(* Schneider Machine Expert - Basic project Controller3(2shkaf), file version 2.4.0.0 *)
(* ProjectInformations: Name=New project *)

HARDWARE
  Cpu 0: TM221CE40T
  ModuleExtensionObject 0: TM3DI32K
  ModuleExtensionObject 1: TM3DI32K
  ModuleExtensionObject 2: TM3DI32K
  ModuleExtensionObject 3: TM3DI32K
  ModuleExtensionObject 4: TM3DI32K
  ModuleExtensionObject 5: TM3DQ32TK
  ModuleExtensionObject 6: TM3DQ32TK
  Cartridge1 0: TMC2SL1
  EthernetConfiguration: NetworkName=M221, IpAllocationMode=FixedAddress, IpAddress=192.168.1.202, SubnetMask=255.255.255.0
  EthernetConfiguration: NetworkName=M221, IpAllocationMode=FixedAddress, IpAddress=0.0.0.0, SubnetMask=0.0.0.0
  SerialLineConfiguration: Baud=Baud19200, Parity=ParityNone, DataBits=DataBits8, StopBits=StopBits1, PhysicalMedium=PhysicalMediumRs485, TransmissionMode=TransmissionModeModbusRtu, SlaveId=1, Addressing=MasterAddressing
  MastTask: UsePeriodScanMode=false, PeriodScan=100
  FastTask: Period=255
  CpuBehavior: StartingMode=StartAutoRunForced, AutoSaveRamOnEeprom=true, WatchdogPeriod=250

SYMBOLS  (address, symbol, comment, settings)
  %M0       SMS  "0_3"
  %TM0        [Preset=3, Base=OneSecond]
  %TM1        [Preset=3, Base=OneSecond]
  %TM2        [Preset=3, Base=OneSecond]
  %TM3        [Preset=3, Base=OneSecond]
  %TM4        [Preset=3, Base=OneSecond]
  %TM5        [Preset=3, Base=OneSecond]
  %TM6        [Preset=3, Base=OneSecond]
  %TM7        [Preset=3, Base=OneSecond]
  %TM8        [Preset=3, Base=OneSecond]
  %TM9        [Preset=3, Base=OneSecond]
  %TM10       [Preset=3, Base=OneSecond]
  %TM11       [Preset=3, Base=OneSecond]
  %TM12       [Preset=3, Base=OneSecond]
  %TM13       [Preset=3, Base=OneSecond]
  %TM14       [Preset=3, Base=OneSecond]
  %TM15       [Preset=3, Base=OneSecond]
  %TM16       [Preset=3, Base=OneSecond]
  %TM17       [Preset=3, Base=OneSecond]
  %TM18       [Preset=3, Base=OneSecond]
  %TM19       [Preset=3, Base=OneSecond]
  %TM20       [Preset=3, Base=OneSecond]
  %TM21       [Preset=3, Base=OneSecond]
  %TM22       [Preset=3, Base=OneSecond]
  %TM23       [Preset=3, Base=OneSecond]

POU Входы 2.0
  (* SectionNumber=1 *)

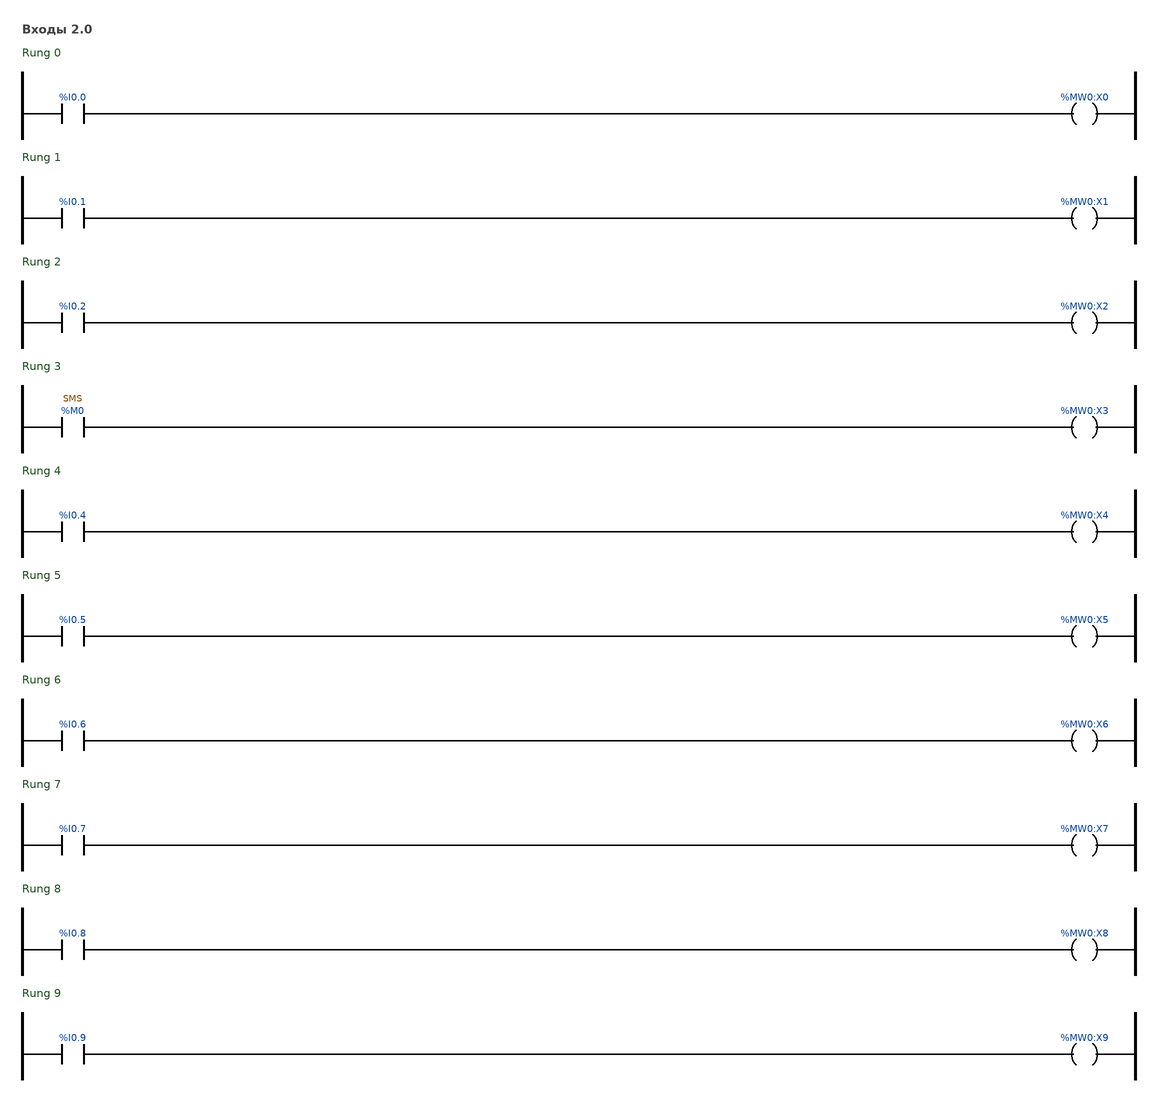

// Rung 0
  LD %I0.0
  ST %MW0:X0
  // as ST:
  //   %MW0:X0 := %I0.0;

// Rung 1
  LD %I0.1
  ST %MW0:X1
  // as ST:
  //   %MW0:X1 := %I0.1;

// Rung 2
  LD %I0.2
  ST %MW0:X2
  // as ST:
  //   %MW0:X2 := %I0.2;

// Rung 3
  LD %M0                  (* SMS *)
  ST %MW0:X3
  // as ST:
  //   %MW0:X3 := SMS;

// Rung 4
  LD %I0.4
  ST %MW0:X4
  // as ST:
  //   %MW0:X4 := %I0.4;

// Rung 5
  LD %I0.5
  ST %MW0:X5
  // as ST:
  //   %MW0:X5 := %I0.5;

// Rung 6
  LD %I0.6
  ST %MW0:X6
  // as ST:
  //   %MW0:X6 := %I0.6;

// Rung 7
  LD %I0.7
  ST %MW0:X7
  // as ST:
  //   %MW0:X7 := %I0.7;

// Rung 8
  LD %I0.8
  ST %MW0:X8
  // as ST:
  //   %MW0:X8 := %I0.8;

// Rung 9
  LD %I0.9
  ST %MW0:X9
  // as ST:
  //   %MW0:X9 := %I0.9;

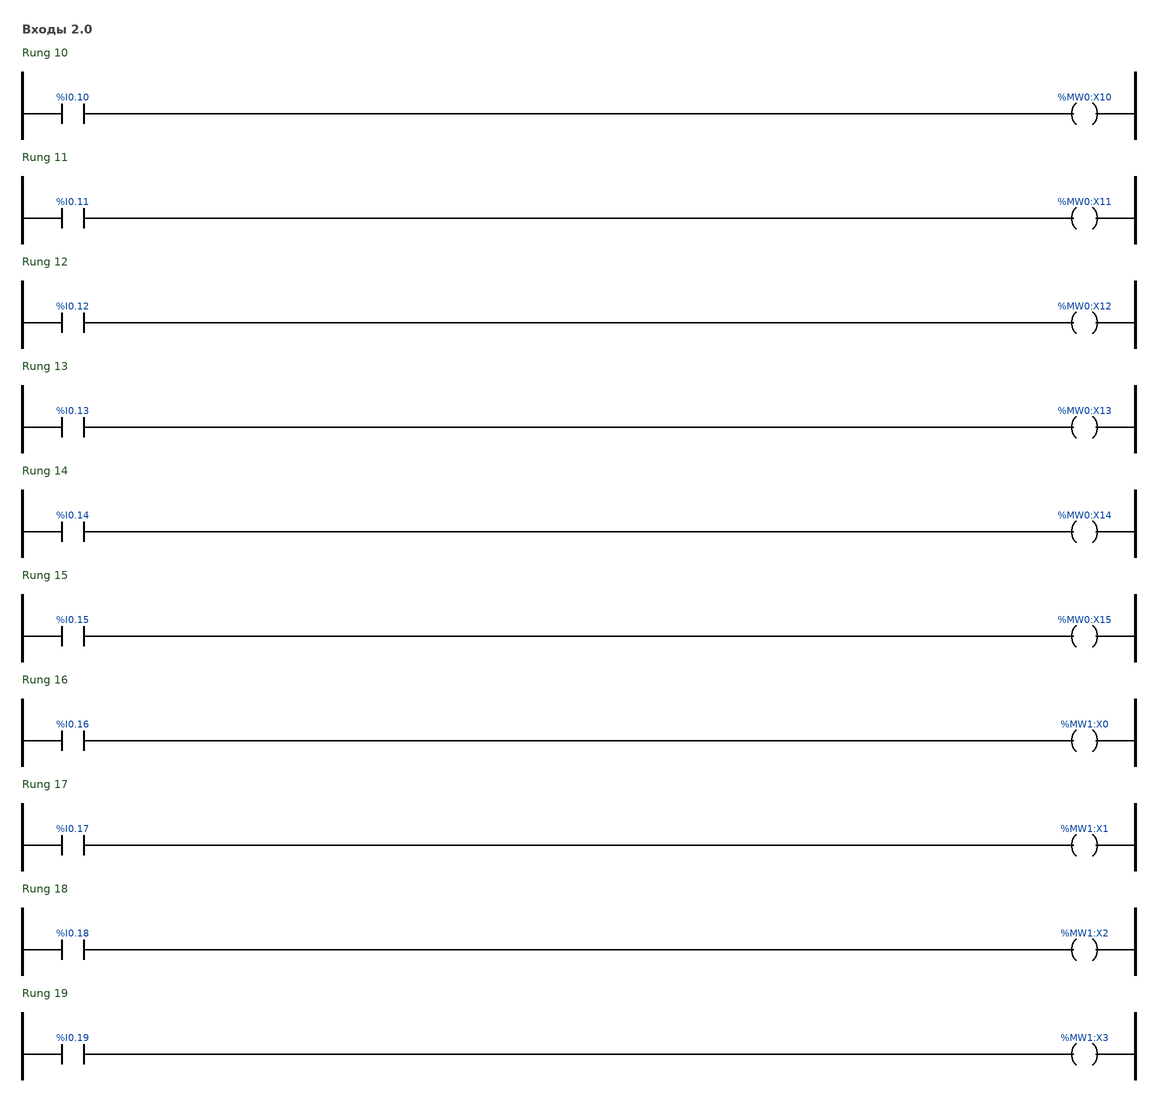

// Rung 10
  LD %I0.10
  ST %MW0:X10
  // as ST:
  //   %MW0:X10 := %I0.10;

// Rung 11
  LD %I0.11
  ST %MW0:X11
  // as ST:
  //   %MW0:X11 := %I0.11;

// Rung 12
  LD %I0.12
  ST %MW0:X12
  // as ST:
  //   %MW0:X12 := %I0.12;

// Rung 13
  LD %I0.13
  ST %MW0:X13
  // as ST:
  //   %MW0:X13 := %I0.13;

// Rung 14
  LD %I0.14
  ST %MW0:X14
  // as ST:
  //   %MW0:X14 := %I0.14;

// Rung 15
  LD %I0.15
  ST %MW0:X15
  // as ST:
  //   %MW0:X15 := %I0.15;

// Rung 16
  LD %I0.16
  ST %MW1:X0
  // as ST:
  //   %MW1:X0 := %I0.16;

// Rung 17
  LD %I0.17
  ST %MW1:X1
  // as ST:
  //   %MW1:X1 := %I0.17;

// Rung 18
  LD %I0.18
  ST %MW1:X2
  // as ST:
  //   %MW1:X2 := %I0.18;

// Rung 19
  LD %I0.19
  ST %MW1:X3
  // as ST:
  //   %MW1:X3 := %I0.19;

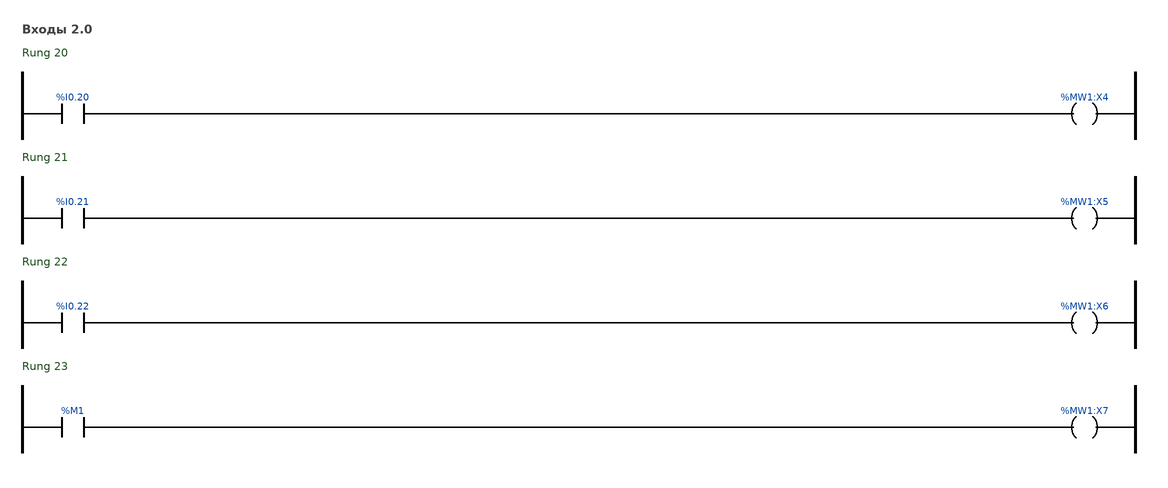

// Rung 20
  LD %I0.20
  ST %MW1:X4
  // as ST:
  //   %MW1:X4 := %I0.20;

// Rung 21
  LD %I0.21
  ST %MW1:X5
  // as ST:
  //   %MW1:X5 := %I0.21;

// Rung 22
  LD %I0.22
  ST %MW1:X6
  // as ST:
  //   %MW1:X6 := %I0.22;

// Rung 23
  LD %M1
  ST %MW1:X7
  // as ST:
  //   %MW1:X7 := %M1;

POU Входы 2.1
  (* SectionNumber=2 *)

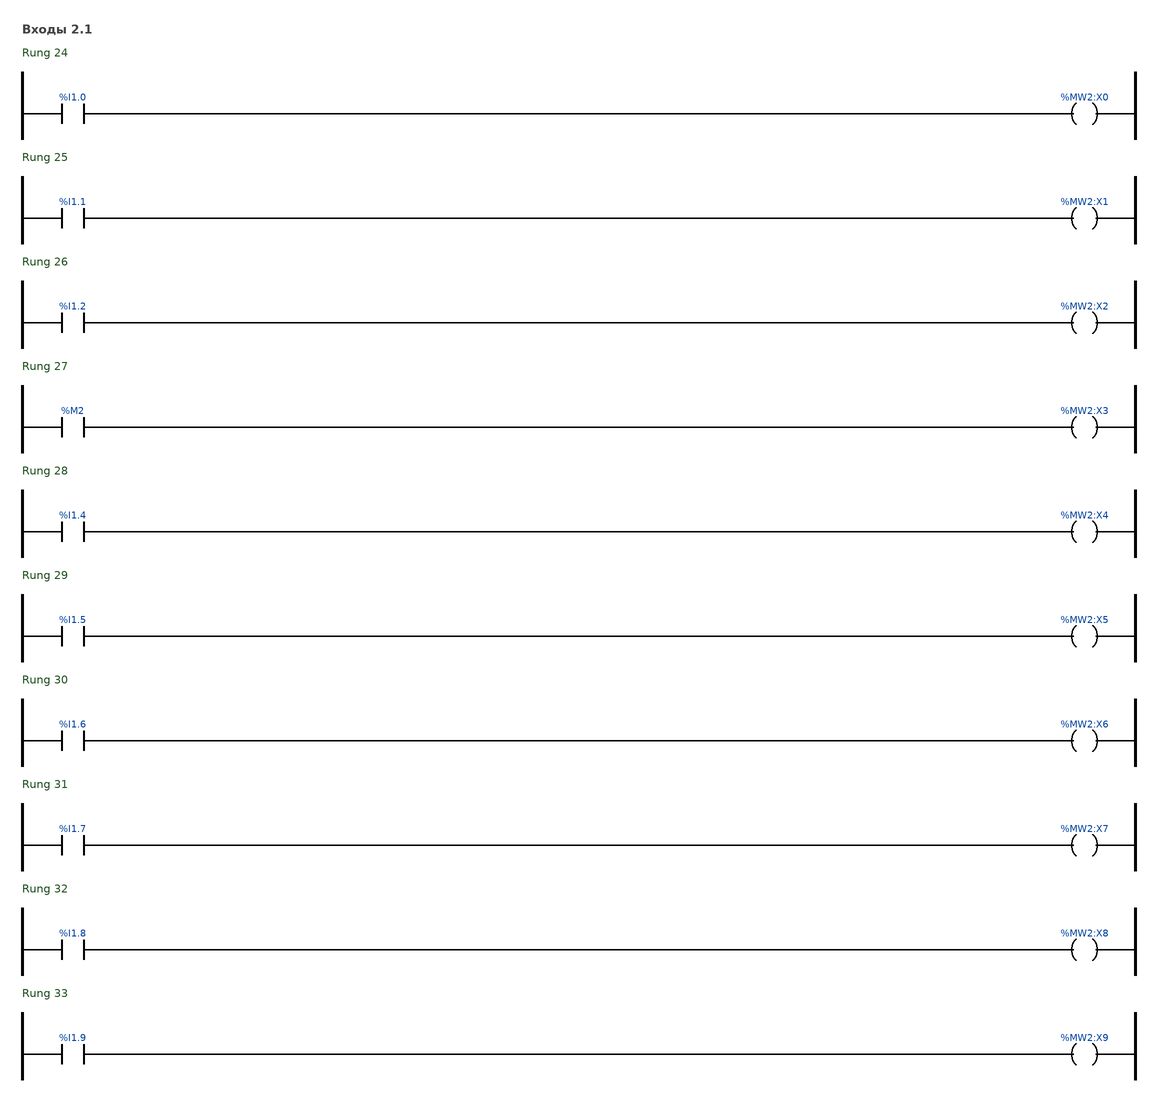

// Rung 24
  LD %I1.0
  ST %MW2:X0
  // as ST:
  //   %MW2:X0 := %I1.0;

// Rung 25
  LD %I1.1
  ST %MW2:X1
  // as ST:
  //   %MW2:X1 := %I1.1;

// Rung 26
  LD %I1.2
  ST %MW2:X2
  // as ST:
  //   %MW2:X2 := %I1.2;

// Rung 27
  LD %M2
  ST %MW2:X3
  // as ST:
  //   %MW2:X3 := %M2;

// Rung 28
  LD %I1.4
  ST %MW2:X4
  // as ST:
  //   %MW2:X4 := %I1.4;

// Rung 29
  LD %I1.5
  ST %MW2:X5
  // as ST:
  //   %MW2:X5 := %I1.5;

// Rung 30
  LD %I1.6
  ST %MW2:X6
  // as ST:
  //   %MW2:X6 := %I1.6;

// Rung 31
  LD %I1.7
  ST %MW2:X7
  // as ST:
  //   %MW2:X7 := %I1.7;

// Rung 32
  LD %I1.8
  ST %MW2:X8
  // as ST:
  //   %MW2:X8 := %I1.8;

// Rung 33
  LD %I1.9
  ST %MW2:X9
  // as ST:
  //   %MW2:X9 := %I1.9;

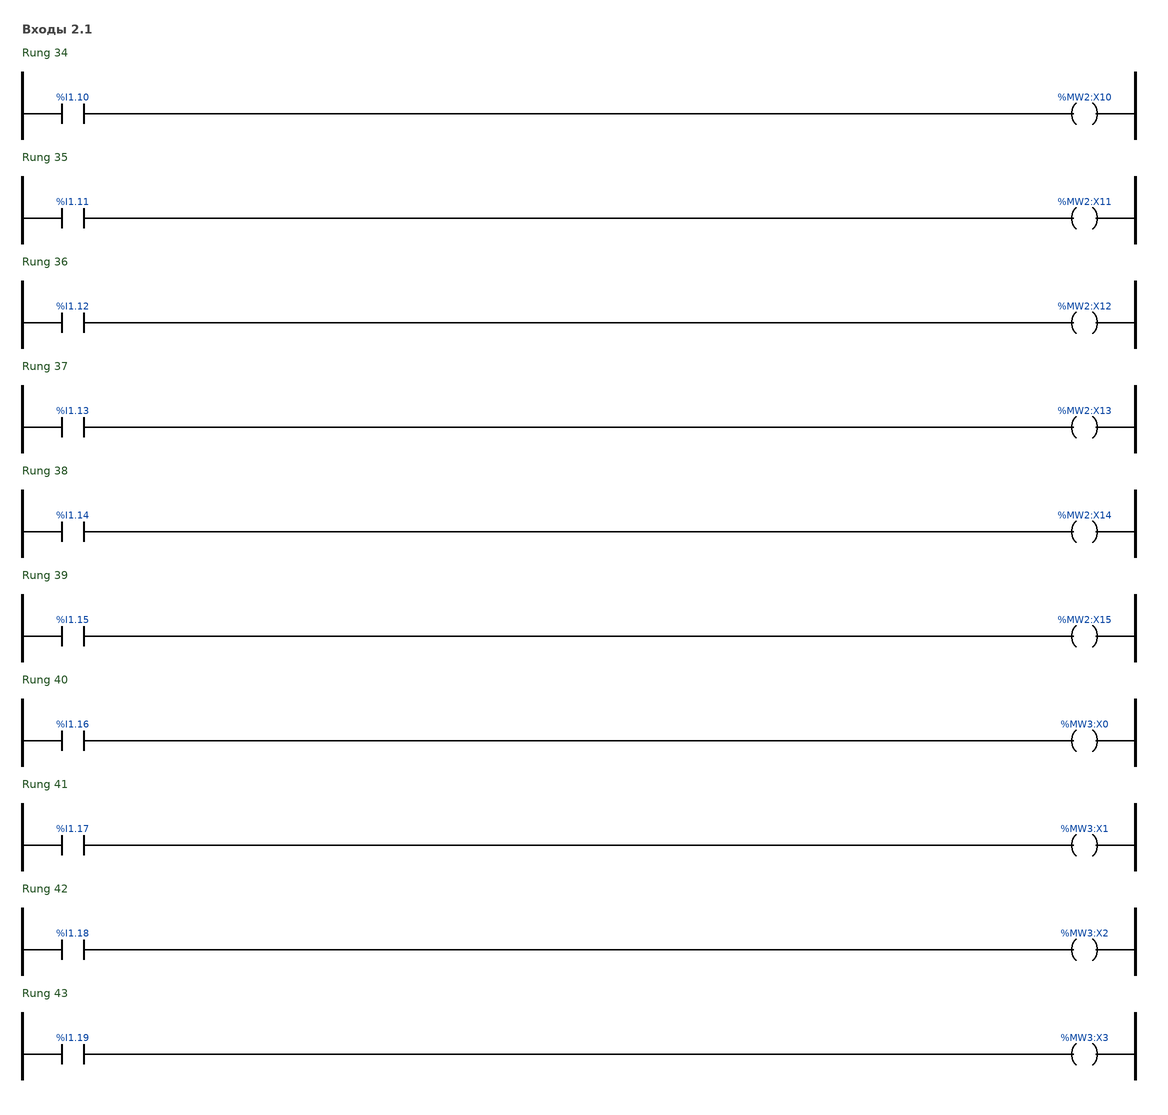

// Rung 34
  LD %I1.10
  ST %MW2:X10
  // as ST:
  //   %MW2:X10 := %I1.10;

// Rung 35
  LD %I1.11
  ST %MW2:X11
  // as ST:
  //   %MW2:X11 := %I1.11;

// Rung 36
  LD %I1.12
  ST %MW2:X12
  // as ST:
  //   %MW2:X12 := %I1.12;

// Rung 37
  LD %I1.13
  ST %MW2:X13
  // as ST:
  //   %MW2:X13 := %I1.13;

// Rung 38
  LD %I1.14
  ST %MW2:X14
  // as ST:
  //   %MW2:X14 := %I1.14;

// Rung 39
  LD %I1.15
  ST %MW2:X15
  // as ST:
  //   %MW2:X15 := %I1.15;

// Rung 40
  LD %I1.16
  ST %MW3:X0
  // as ST:
  //   %MW3:X0 := %I1.16;

// Rung 41
  LD %I1.17
  ST %MW3:X1
  // as ST:
  //   %MW3:X1 := %I1.17;

// Rung 42
  LD %I1.18
  ST %MW3:X2
  // as ST:
  //   %MW3:X2 := %I1.18;

// Rung 43
  LD %I1.19
  ST %MW3:X3
  // as ST:
  //   %MW3:X3 := %I1.19;

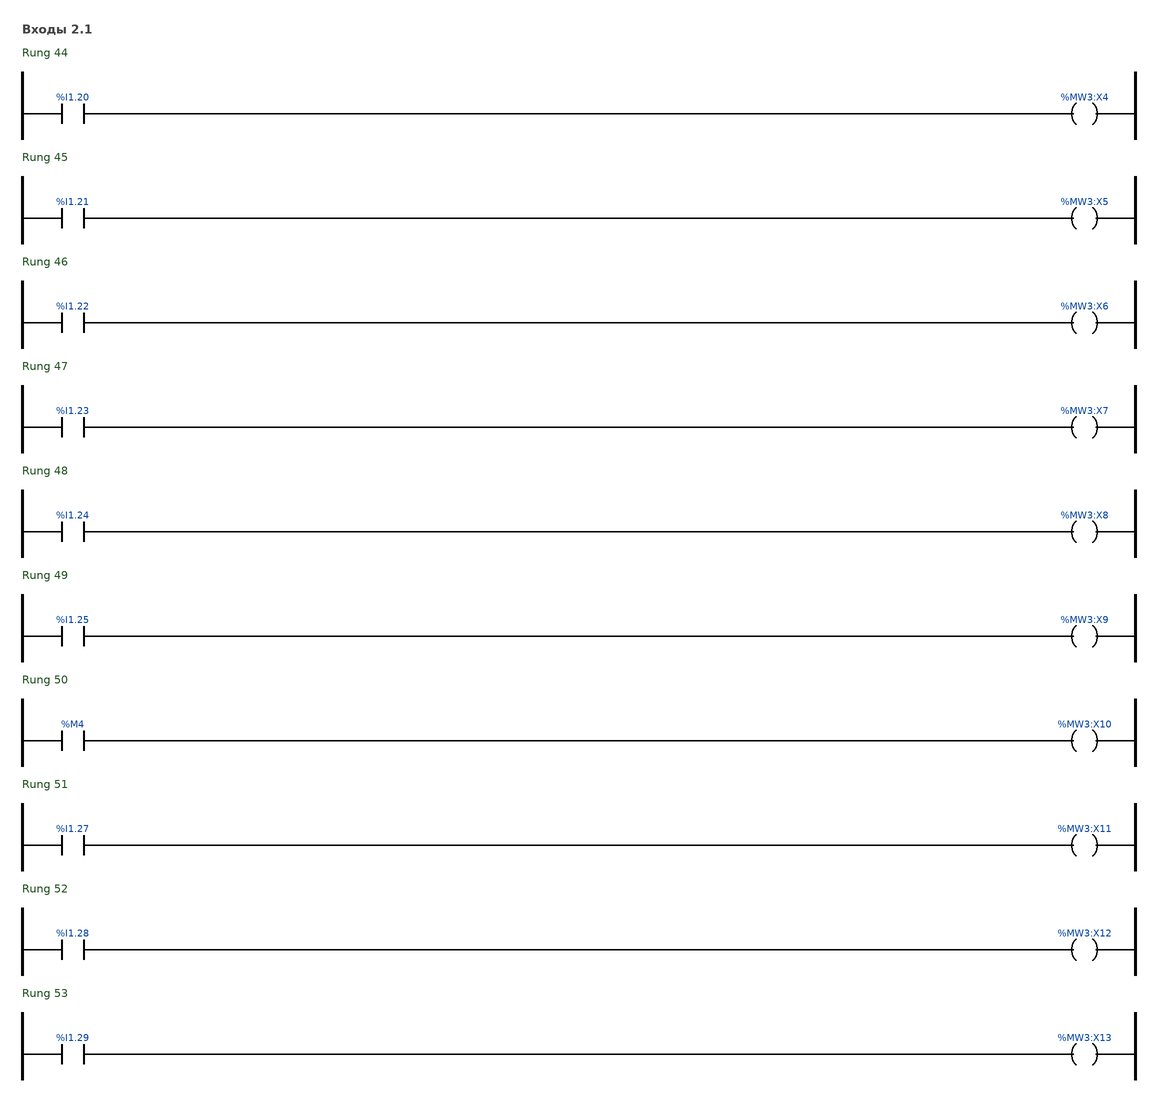

// Rung 44
  LD %I1.20
  ST %MW3:X4
  // as ST:
  //   %MW3:X4 := %I1.20;

// Rung 45
  LD %I1.21
  ST %MW3:X5
  // as ST:
  //   %MW3:X5 := %I1.21;

// Rung 46
  LD %I1.22
  ST %MW3:X6
  // as ST:
  //   %MW3:X6 := %I1.22;

// Rung 47
  LD %I1.23
  ST %MW3:X7
  // as ST:
  //   %MW3:X7 := %I1.23;

// Rung 48
  LD %I1.24
  ST %MW3:X8
  // as ST:
  //   %MW3:X8 := %I1.24;

// Rung 49
  LD %I1.25
  ST %MW3:X9
  // as ST:
  //   %MW3:X9 := %I1.25;

// Rung 50
  LD %M4
  ST %MW3:X10
  // as ST:
  //   %MW3:X10 := %M4;

// Rung 51
  LD %I1.27
  ST %MW3:X11
  // as ST:
  //   %MW3:X11 := %I1.27;

// Rung 52
  LD %I1.28
  ST %MW3:X12
  // as ST:
  //   %MW3:X12 := %I1.28;

// Rung 53
  LD %I1.29
  ST %MW3:X13
  // as ST:
  //   %MW3:X13 := %I1.29;

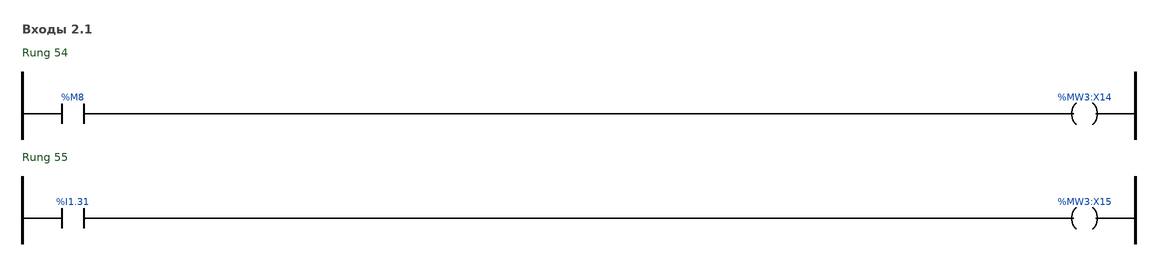

// Rung 54
  LD %M8
  ST %MW3:X14
  // as ST:
  //   %MW3:X14 := %M8;

// Rung 55
  LD %I1.31
  ST %MW3:X15
  // as ST:
  //   %MW3:X15 := %I1.31;

POU Входы 2.2
  (* SectionNumber=3 *)

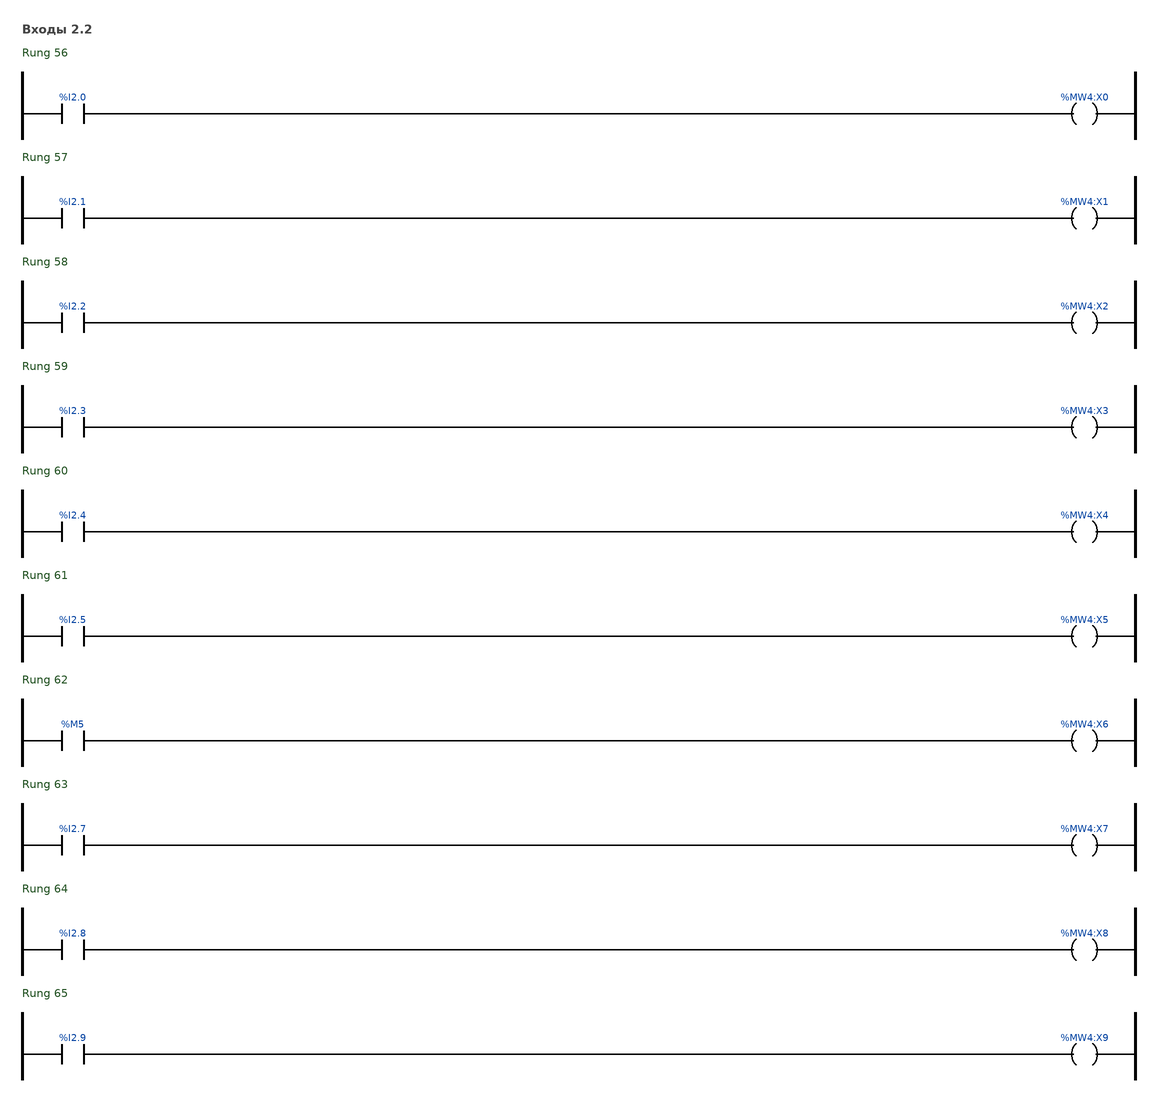

// Rung 56
  LD %I2.0
  ST %MW4:X0
  // as ST:
  //   %MW4:X0 := %I2.0;

// Rung 57
  LD %I2.1
  ST %MW4:X1
  // as ST:
  //   %MW4:X1 := %I2.1;

// Rung 58
  LD %I2.2
  ST %MW4:X2
  // as ST:
  //   %MW4:X2 := %I2.2;

// Rung 59
  LD %I2.3
  ST %MW4:X3
  // as ST:
  //   %MW4:X3 := %I2.3;

// Rung 60
  LD %I2.4
  ST %MW4:X4
  // as ST:
  //   %MW4:X4 := %I2.4;

// Rung 61
  LD %I2.5
  ST %MW4:X5
  // as ST:
  //   %MW4:X5 := %I2.5;

// Rung 62
  LD %M5
  ST %MW4:X6
  // as ST:
  //   %MW4:X6 := %M5;

// Rung 63
  LD %I2.7
  ST %MW4:X7
  // as ST:
  //   %MW4:X7 := %I2.7;

// Rung 64
  LD %I2.8
  ST %MW4:X8
  // as ST:
  //   %MW4:X8 := %I2.8;

// Rung 65
  LD %I2.9
  ST %MW4:X9
  // as ST:
  //   %MW4:X9 := %I2.9;

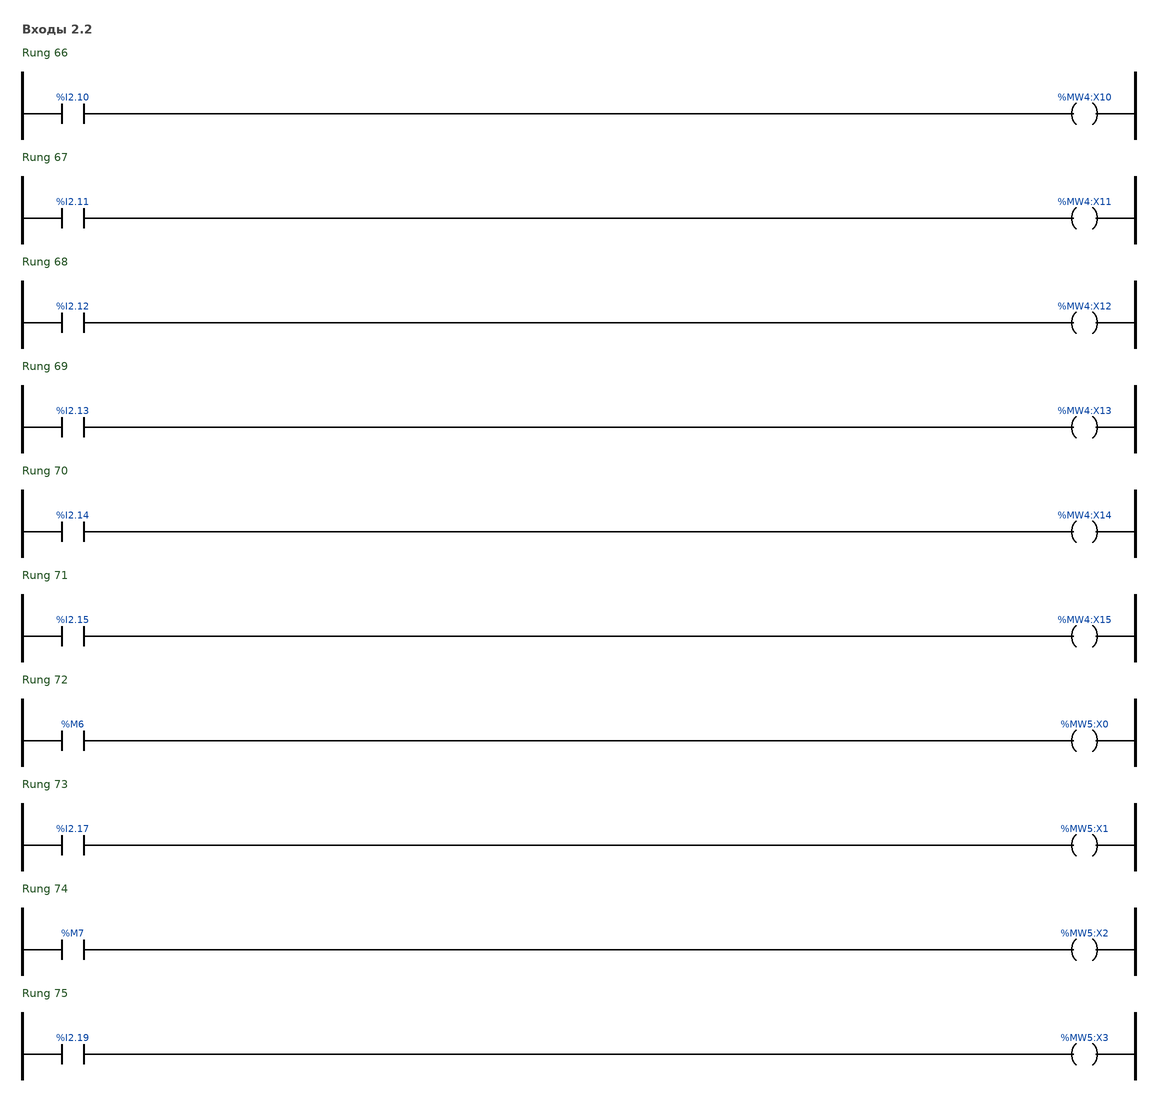

// Rung 66
  LD %I2.10
  ST %MW4:X10
  // as ST:
  //   %MW4:X10 := %I2.10;

// Rung 67
  LD %I2.11
  ST %MW4:X11
  // as ST:
  //   %MW4:X11 := %I2.11;

// Rung 68
  LD %I2.12
  ST %MW4:X12
  // as ST:
  //   %MW4:X12 := %I2.12;

// Rung 69
  LD %I2.13
  ST %MW4:X13
  // as ST:
  //   %MW4:X13 := %I2.13;

// Rung 70
  LD %I2.14
  ST %MW4:X14
  // as ST:
  //   %MW4:X14 := %I2.14;

// Rung 71
  LD %I2.15
  ST %MW4:X15
  // as ST:
  //   %MW4:X15 := %I2.15;

// Rung 72
  LD %M6
  ST %MW5:X0
  // as ST:
  //   %MW5:X0 := %M6;

// Rung 73
  LD %I2.17
  ST %MW5:X1
  // as ST:
  //   %MW5:X1 := %I2.17;

// Rung 74
  LD %M7
  ST %MW5:X2
  // as ST:
  //   %MW5:X2 := %M7;

// Rung 75
  LD %I2.19
  ST %MW5:X3
  // as ST:
  //   %MW5:X3 := %I2.19;

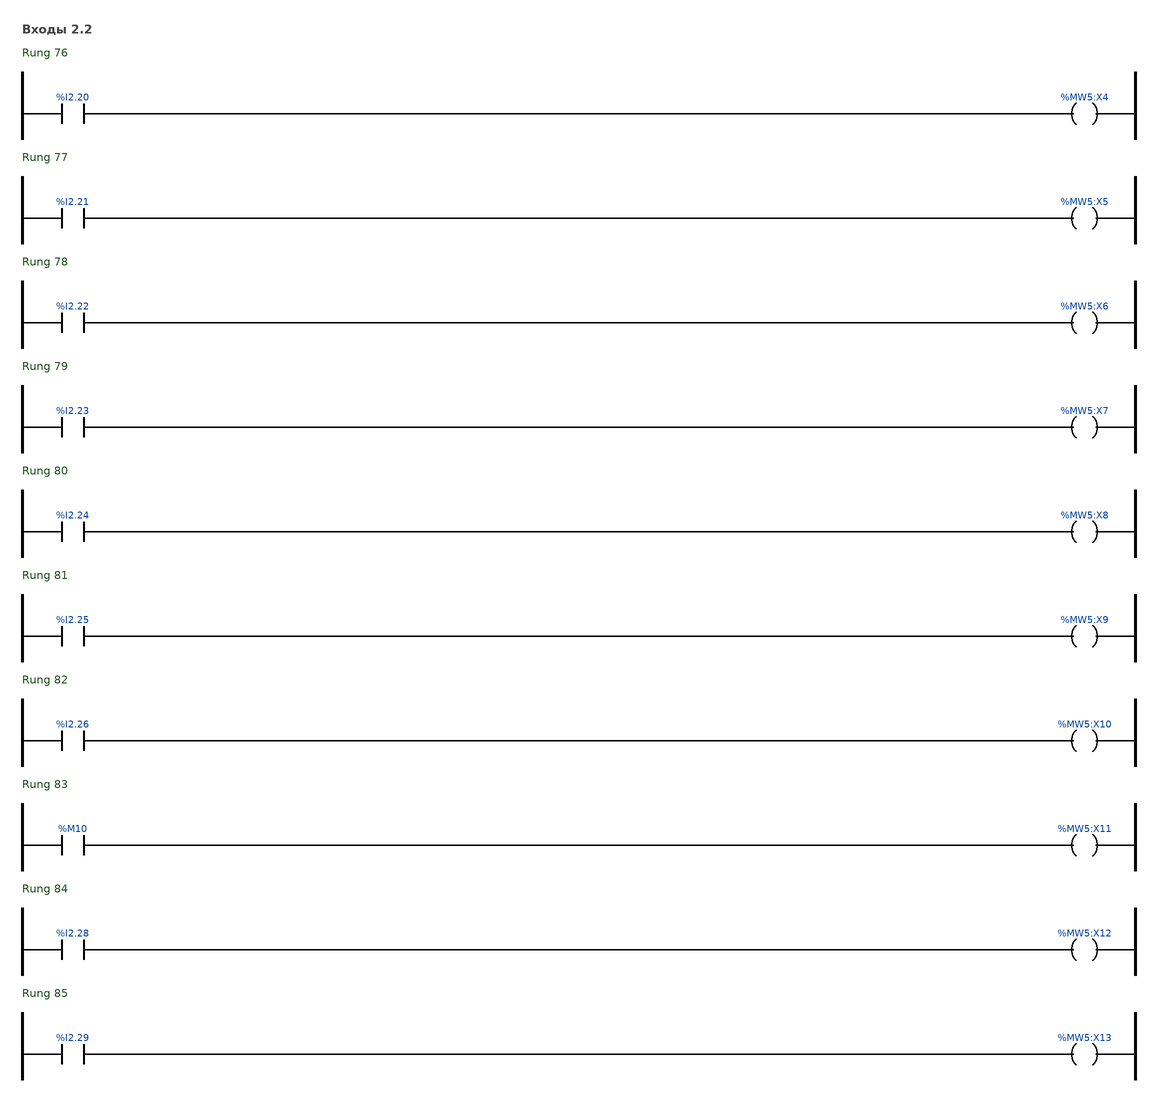

// Rung 76
  LD %I2.20
  ST %MW5:X4
  // as ST:
  //   %MW5:X4 := %I2.20;

// Rung 77
  LD %I2.21
  ST %MW5:X5
  // as ST:
  //   %MW5:X5 := %I2.21;

// Rung 78
  LD %I2.22
  ST %MW5:X6
  // as ST:
  //   %MW5:X6 := %I2.22;

// Rung 79
  LD %I2.23
  ST %MW5:X7
  // as ST:
  //   %MW5:X7 := %I2.23;

// Rung 80
  LD %I2.24
  ST %MW5:X8
  // as ST:
  //   %MW5:X8 := %I2.24;

// Rung 81
  LD %I2.25
  ST %MW5:X9
  // as ST:
  //   %MW5:X9 := %I2.25;

// Rung 82
  LD %I2.26
  ST %MW5:X10
  // as ST:
  //   %MW5:X10 := %I2.26;

// Rung 83
  LD %M10
  ST %MW5:X11
  // as ST:
  //   %MW5:X11 := %M10;

// Rung 84
  LD %I2.28
  ST %MW5:X12
  // as ST:
  //   %MW5:X12 := %I2.28;

// Rung 85
  LD %I2.29
  ST %MW5:X13
  // as ST:
  //   %MW5:X13 := %I2.29;

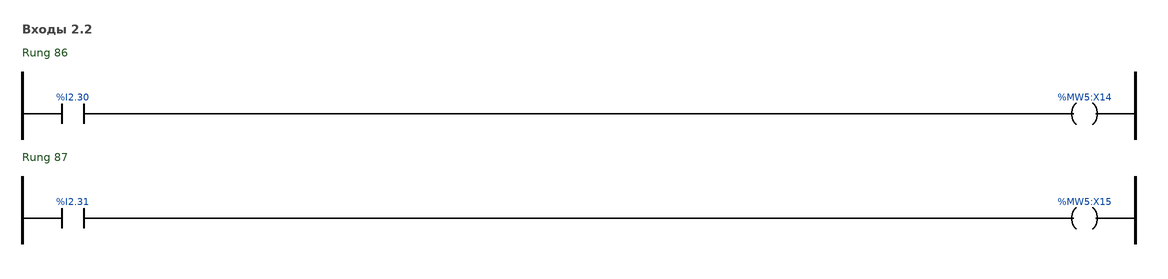

// Rung 86
  LD %I2.30
  ST %MW5:X14
  // as ST:
  //   %MW5:X14 := %I2.30;

// Rung 87
  LD %I2.31
  ST %MW5:X15
  // as ST:
  //   %MW5:X15 := %I2.31;

POU Входы 2.3
  (* SectionNumber=4 *)

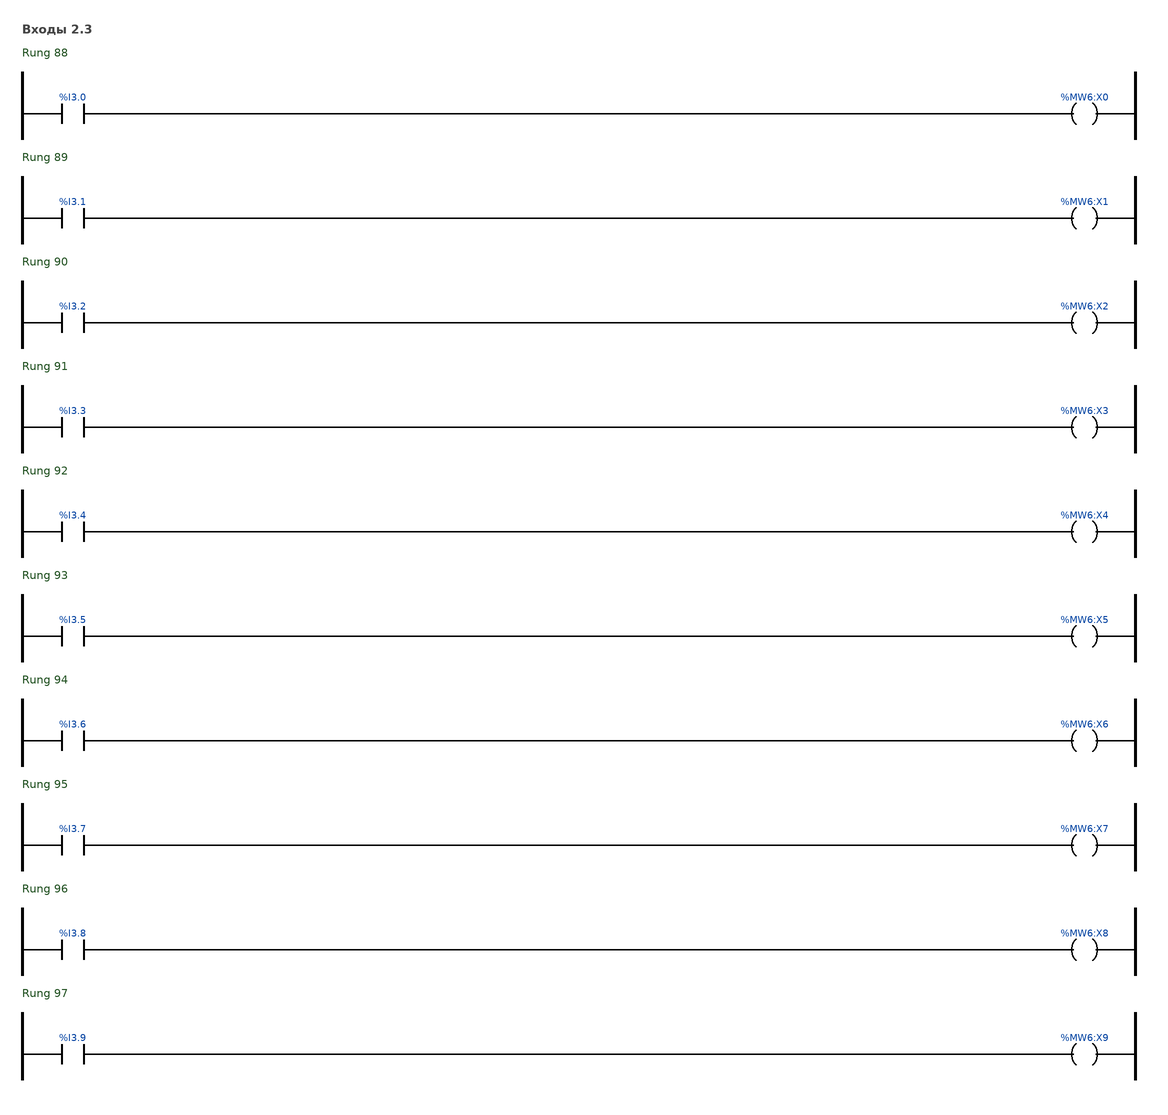

// Rung 88
  LD %I3.0
  ST %MW6:X0
  // as ST:
  //   %MW6:X0 := %I3.0;

// Rung 89
  LD %I3.1
  ST %MW6:X1
  // as ST:
  //   %MW6:X1 := %I3.1;

// Rung 90
  LD %I3.2
  ST %MW6:X2
  // as ST:
  //   %MW6:X2 := %I3.2;

// Rung 91
  LD %I3.3
  ST %MW6:X3
  // as ST:
  //   %MW6:X3 := %I3.3;

// Rung 92
  LD %I3.4
  ST %MW6:X4
  // as ST:
  //   %MW6:X4 := %I3.4;

// Rung 93
  LD %I3.5
  ST %MW6:X5
  // as ST:
  //   %MW6:X5 := %I3.5;

// Rung 94
  LD %I3.6
  ST %MW6:X6
  // as ST:
  //   %MW6:X6 := %I3.6;

// Rung 95
  LD %I3.7
  ST %MW6:X7
  // as ST:
  //   %MW6:X7 := %I3.7;

// Rung 96
  LD %I3.8
  ST %MW6:X8
  // as ST:
  //   %MW6:X8 := %I3.8;

// Rung 97
  LD %I3.9
  ST %MW6:X9
  // as ST:
  //   %MW6:X9 := %I3.9;

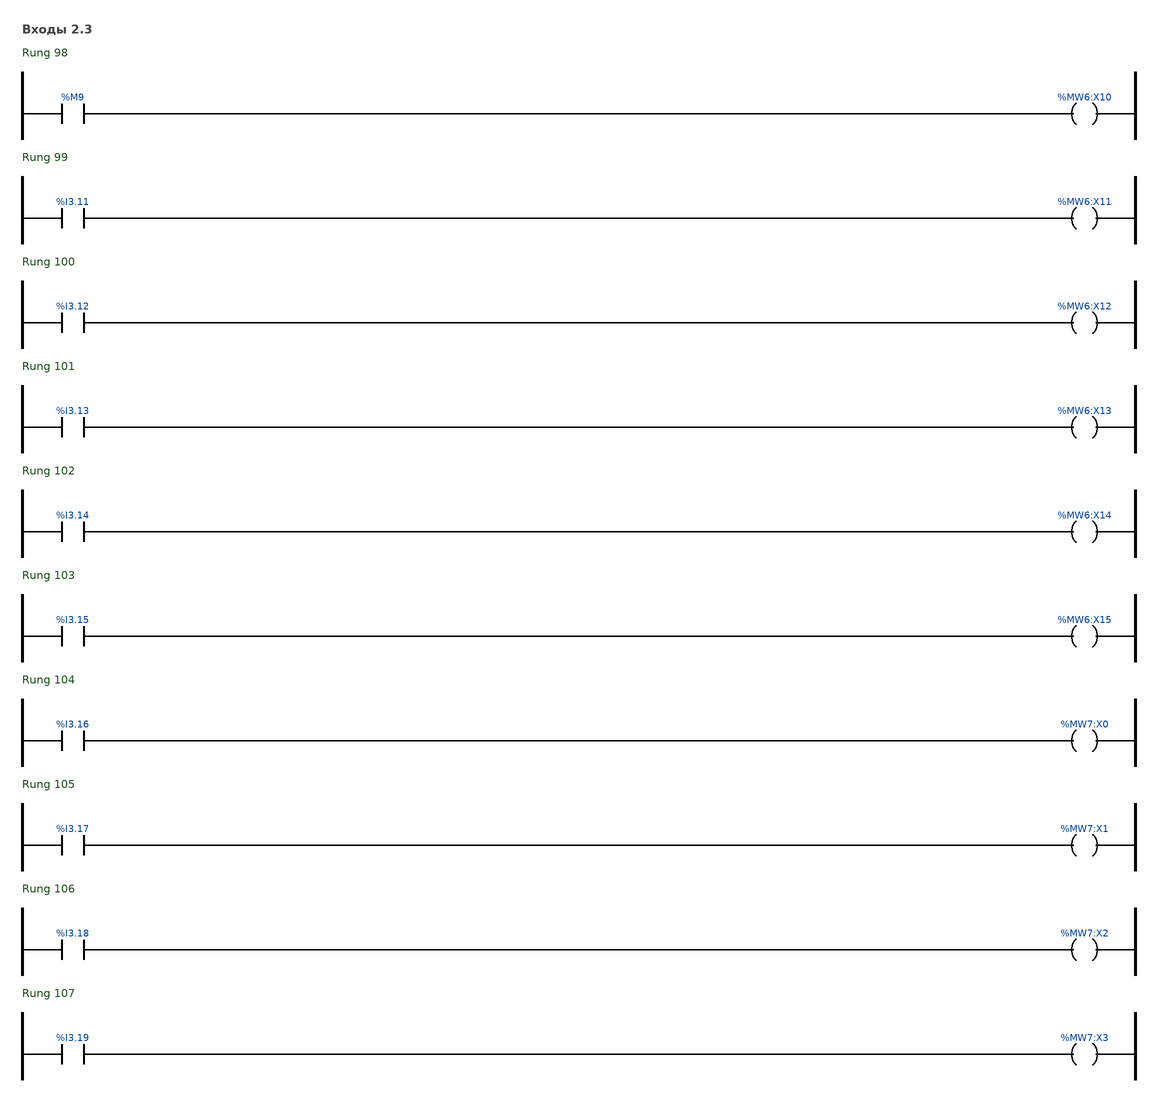

// Rung 98
  LD %M9
  ST %MW6:X10
  // as ST:
  //   %MW6:X10 := %M9;

// Rung 99
  LD %I3.11
  ST %MW6:X11
  // as ST:
  //   %MW6:X11 := %I3.11;

// Rung 100
  LD %I3.12
  ST %MW6:X12
  // as ST:
  //   %MW6:X12 := %I3.12;

// Rung 101
  LD %I3.13
  ST %MW6:X13
  // as ST:
  //   %MW6:X13 := %I3.13;

// Rung 102
  LD %I3.14
  ST %MW6:X14
  // as ST:
  //   %MW6:X14 := %I3.14;

// Rung 103
  LD %I3.15
  ST %MW6:X15
  // as ST:
  //   %MW6:X15 := %I3.15;

// Rung 104
  LD %I3.16
  ST %MW7:X0
  // as ST:
  //   %MW7:X0 := %I3.16;

// Rung 105
  LD %I3.17
  ST %MW7:X1
  // as ST:
  //   %MW7:X1 := %I3.17;

// Rung 106
  LD %I3.18
  ST %MW7:X2
  // as ST:
  //   %MW7:X2 := %I3.18;

// Rung 107
  LD %I3.19
  ST %MW7:X3
  // as ST:
  //   %MW7:X3 := %I3.19;

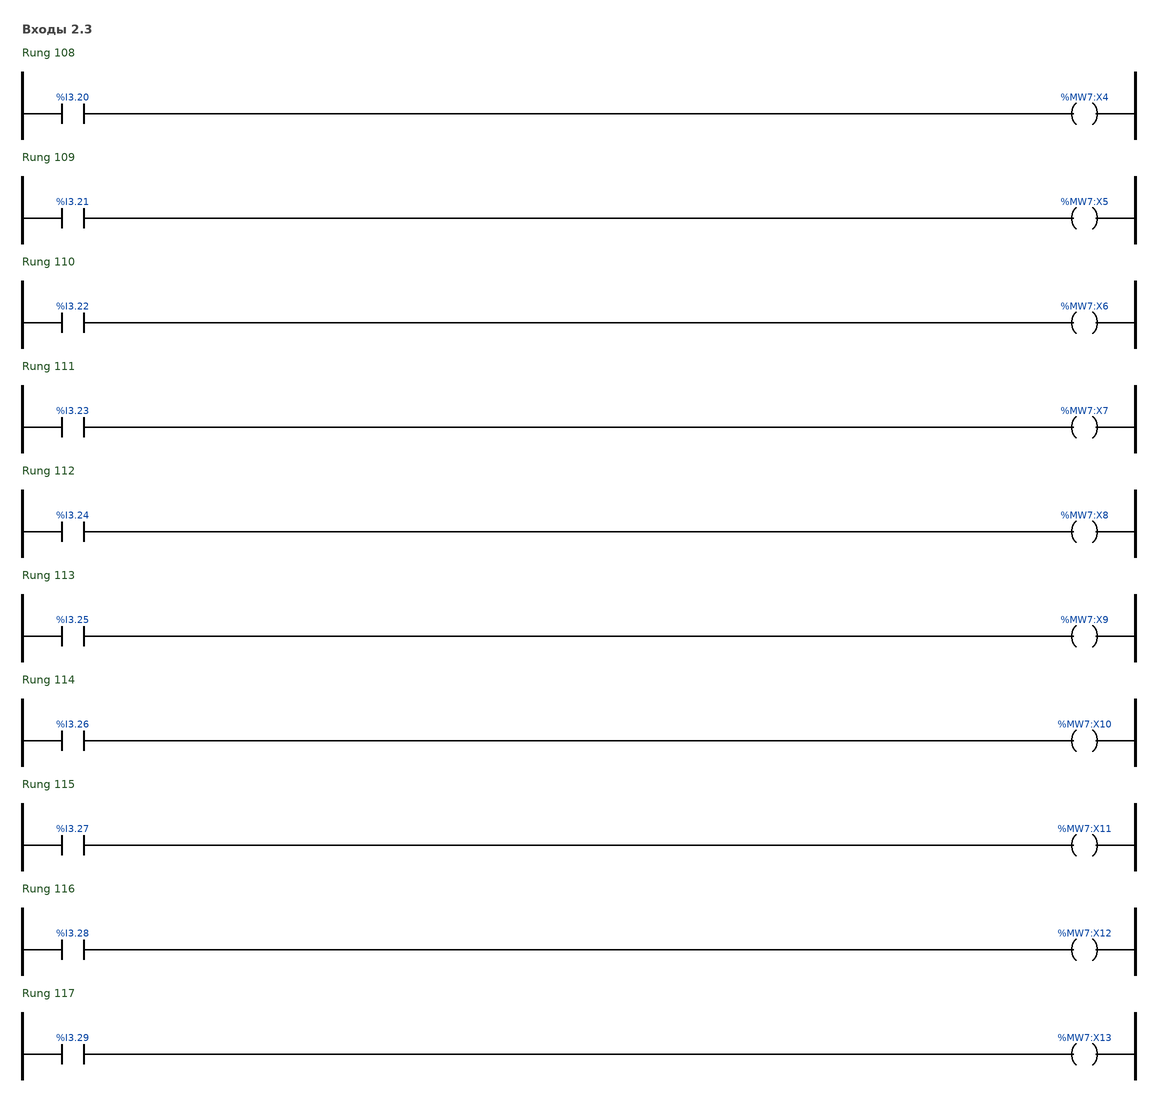

// Rung 108
  LD %I3.20
  ST %MW7:X4
  // as ST:
  //   %MW7:X4 := %I3.20;

// Rung 109
  LD %I3.21
  ST %MW7:X5
  // as ST:
  //   %MW7:X5 := %I3.21;

// Rung 110
  LD %I3.22
  ST %MW7:X6
  // as ST:
  //   %MW7:X6 := %I3.22;

// Rung 111
  LD %I3.23
  ST %MW7:X7
  // as ST:
  //   %MW7:X7 := %I3.23;

// Rung 112
  LD %I3.24
  ST %MW7:X8
  // as ST:
  //   %MW7:X8 := %I3.24;

// Rung 113
  LD %I3.25
  ST %MW7:X9
  // as ST:
  //   %MW7:X9 := %I3.25;

// Rung 114
  LD %I3.26
  ST %MW7:X10
  // as ST:
  //   %MW7:X10 := %I3.26;

// Rung 115
  LD %I3.27
  ST %MW7:X11
  // as ST:
  //   %MW7:X11 := %I3.27;

// Rung 116
  LD %I3.28
  ST %MW7:X12
  // as ST:
  //   %MW7:X12 := %I3.28;

// Rung 117
  LD %I3.29
  ST %MW7:X13
  // as ST:
  //   %MW7:X13 := %I3.29;

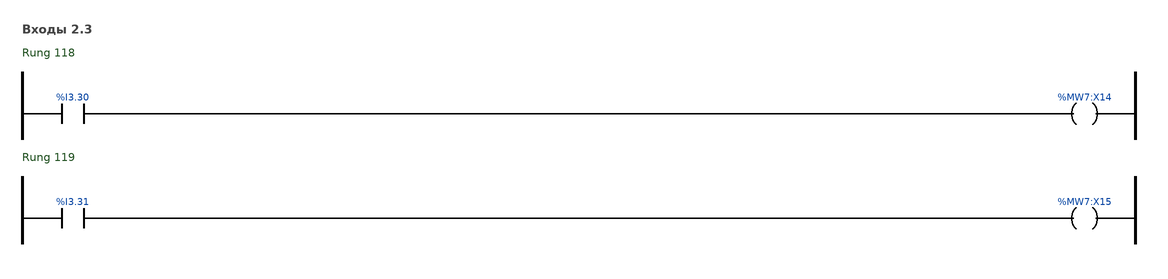

// Rung 118
  LD %I3.30
  ST %MW7:X14
  // as ST:
  //   %MW7:X14 := %I3.30;

// Rung 119
  LD %I3.31
  ST %MW7:X15
  // as ST:
  //   %MW7:X15 := %I3.31;

POU Входы 2.4
  (* SectionNumber=5 *)

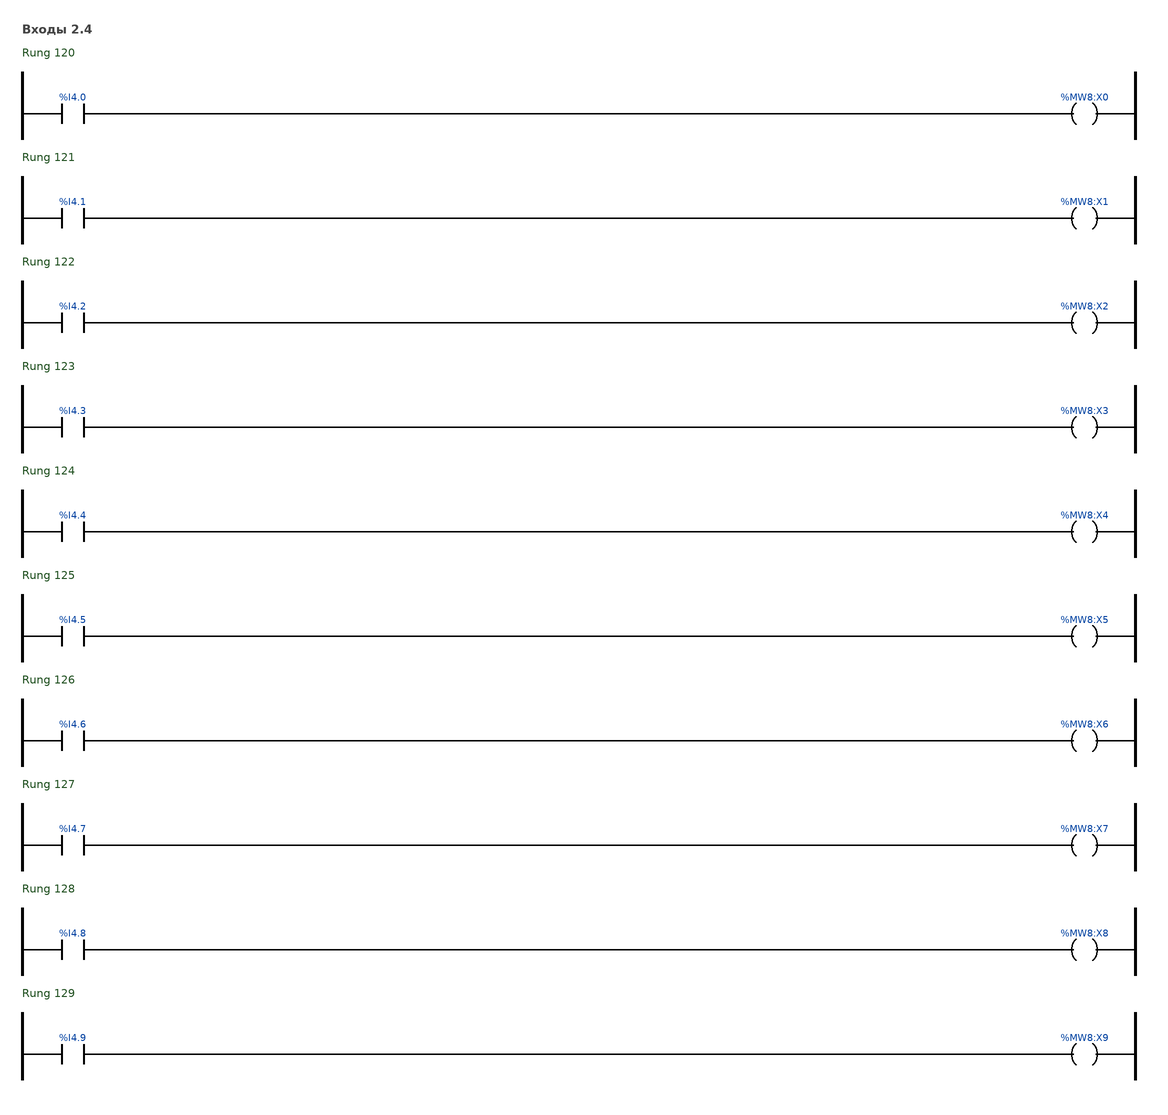

// Rung 120
  LD %I4.0
  ST %MW8:X0
  // as ST:
  //   %MW8:X0 := %I4.0;

// Rung 121
  LD %I4.1
  ST %MW8:X1
  // as ST:
  //   %MW8:X1 := %I4.1;

// Rung 122
  LD %I4.2
  ST %MW8:X2
  // as ST:
  //   %MW8:X2 := %I4.2;

// Rung 123
  LD %I4.3
  ST %MW8:X3
  // as ST:
  //   %MW8:X3 := %I4.3;

// Rung 124
  LD %I4.4
  ST %MW8:X4
  // as ST:
  //   %MW8:X4 := %I4.4;

// Rung 125
  LD %I4.5
  ST %MW8:X5
  // as ST:
  //   %MW8:X5 := %I4.5;

// Rung 126
  LD %I4.6
  ST %MW8:X6
  // as ST:
  //   %MW8:X6 := %I4.6;

// Rung 127
  LD %I4.7
  ST %MW8:X7
  // as ST:
  //   %MW8:X7 := %I4.7;

// Rung 128
  LD %I4.8
  ST %MW8:X8
  // as ST:
  //   %MW8:X8 := %I4.8;

// Rung 129
  LD %I4.9
  ST %MW8:X9
  // as ST:
  //   %MW8:X9 := %I4.9;

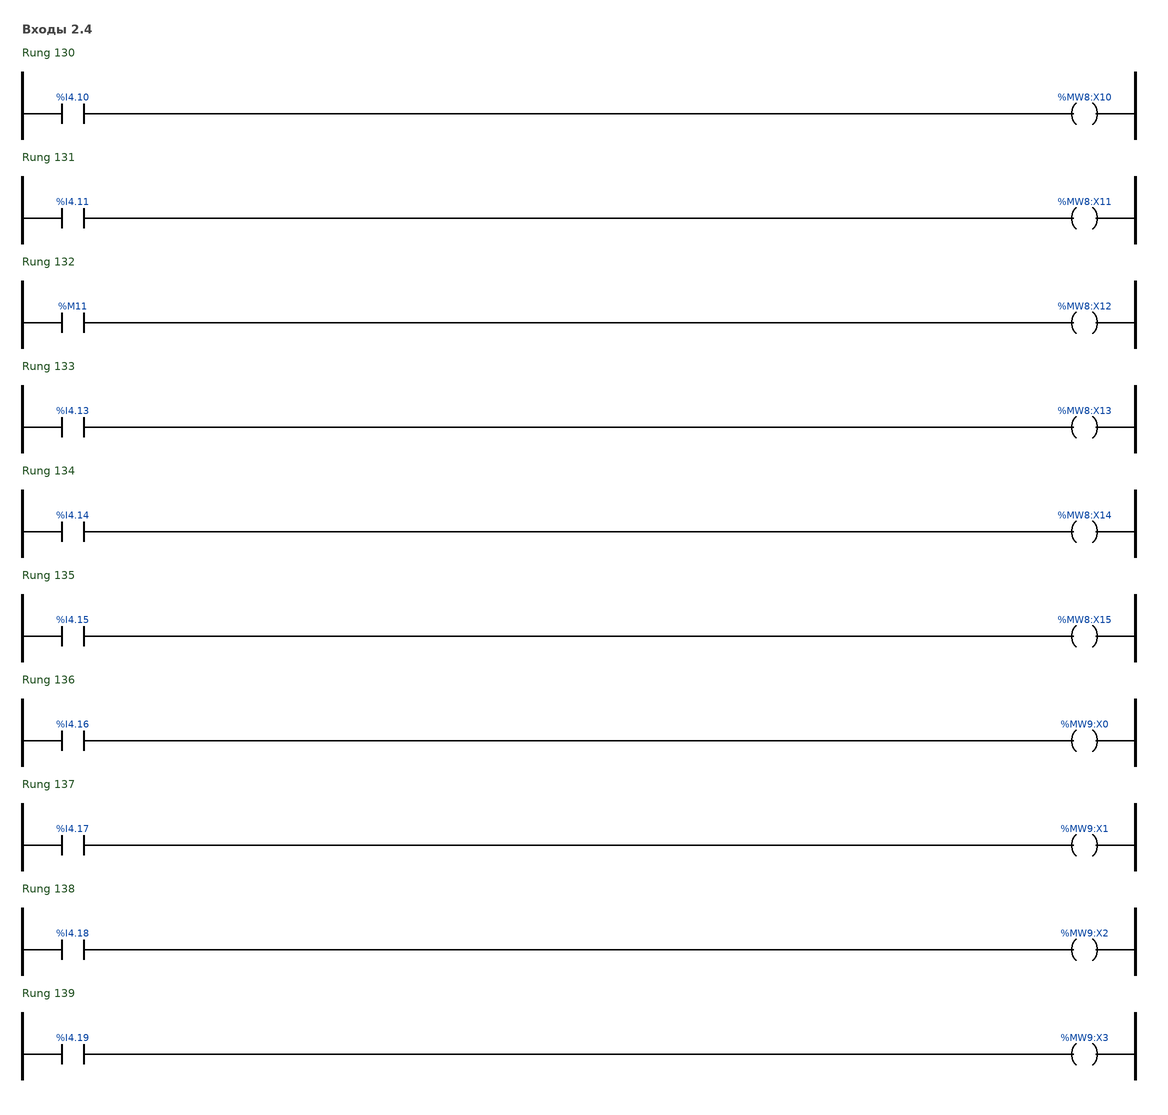

// Rung 130
  LD %I4.10
  ST %MW8:X10
  // as ST:
  //   %MW8:X10 := %I4.10;

// Rung 131
  LD %I4.11
  ST %MW8:X11
  // as ST:
  //   %MW8:X11 := %I4.11;

// Rung 132
  LD %M11
  ST %MW8:X12
  // as ST:
  //   %MW8:X12 := %M11;

// Rung 133
  LD %I4.13
  ST %MW8:X13
  // as ST:
  //   %MW8:X13 := %I4.13;

// Rung 134
  LD %I4.14
  ST %MW8:X14
  // as ST:
  //   %MW8:X14 := %I4.14;

// Rung 135
  LD %I4.15
  ST %MW8:X15
  // as ST:
  //   %MW8:X15 := %I4.15;

// Rung 136
  LD %I4.16
  ST %MW9:X0
  // as ST:
  //   %MW9:X0 := %I4.16;

// Rung 137
  LD %I4.17
  ST %MW9:X1
  // as ST:
  //   %MW9:X1 := %I4.17;

// Rung 138
  LD %I4.18
  ST %MW9:X2
  // as ST:
  //   %MW9:X2 := %I4.18;

// Rung 139
  LD %I4.19
  ST %MW9:X3
  // as ST:
  //   %MW9:X3 := %I4.19;

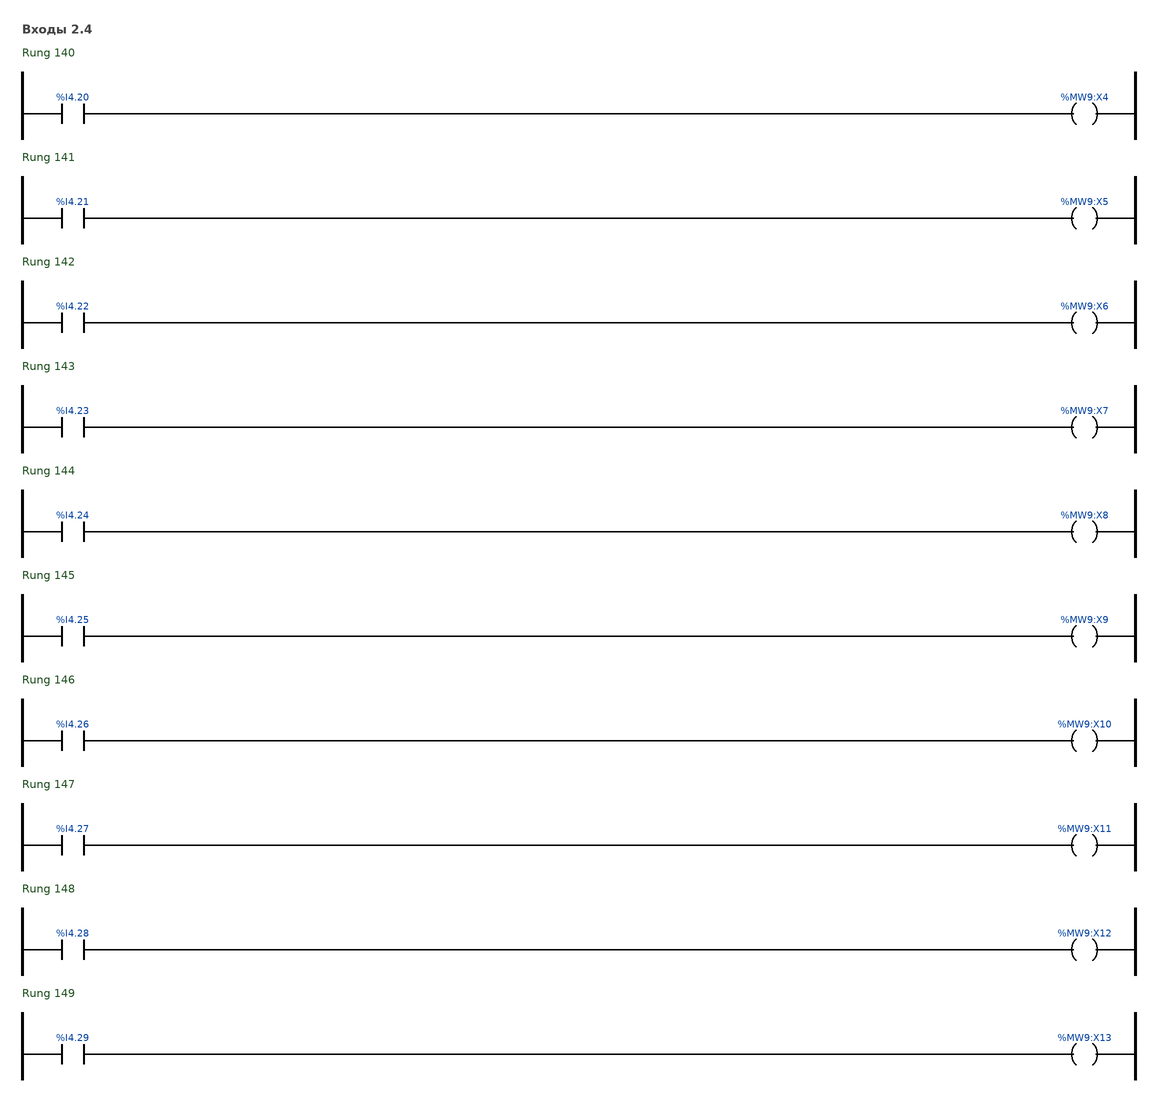

// Rung 140
  LD %I4.20
  ST %MW9:X4
  // as ST:
  //   %MW9:X4 := %I4.20;

// Rung 141
  LD %I4.21
  ST %MW9:X5
  // as ST:
  //   %MW9:X5 := %I4.21;

// Rung 142
  LD %I4.22
  ST %MW9:X6
  // as ST:
  //   %MW9:X6 := %I4.22;

// Rung 143
  LD %I4.23
  ST %MW9:X7
  // as ST:
  //   %MW9:X7 := %I4.23;

// Rung 144
  LD %I4.24
  ST %MW9:X8
  // as ST:
  //   %MW9:X8 := %I4.24;

// Rung 145
  LD %I4.25
  ST %MW9:X9
  // as ST:
  //   %MW9:X9 := %I4.25;

// Rung 146
  LD %I4.26
  ST %MW9:X10
  // as ST:
  //   %MW9:X10 := %I4.26;

// Rung 147
  LD %I4.27
  ST %MW9:X11
  // as ST:
  //   %MW9:X11 := %I4.27;

// Rung 148
  LD %I4.28
  ST %MW9:X12
  // as ST:
  //   %MW9:X12 := %I4.28;

// Rung 149
  LD %I4.29
  ST %MW9:X13
  // as ST:
  //   %MW9:X13 := %I4.29;

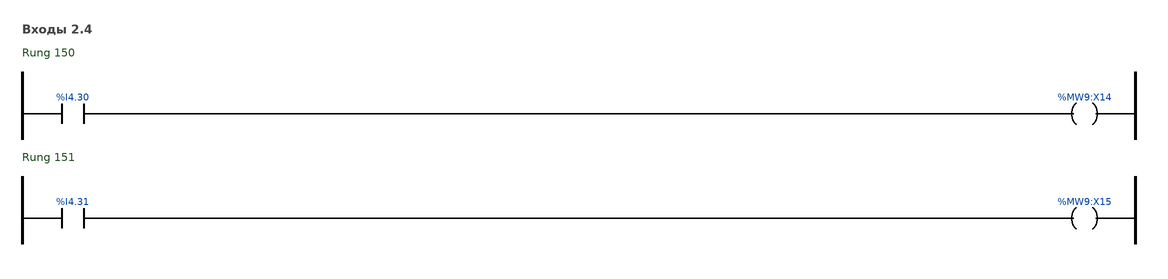

// Rung 150
  LD %I4.30
  ST %MW9:X14
  // as ST:
  //   %MW9:X14 := %I4.30;

// Rung 151
  LD %I4.31
  ST %MW9:X15
  // as ST:
  //   %MW9:X15 := %I4.31;

POU Входы 2.5
  (* SectionNumber=6 *)

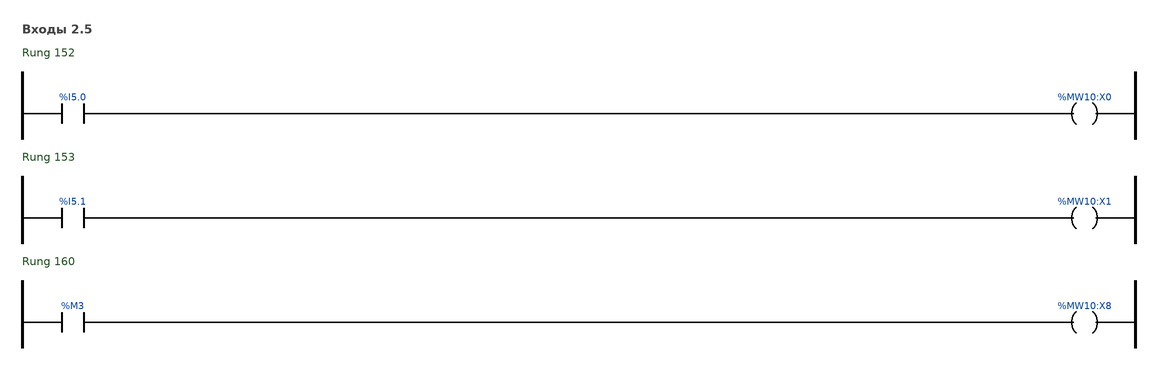

// Rung 152
  LD %I5.0
  ST %MW10:X0
  // as ST:
  //   %MW10:X0 := %I5.0;

// Rung 153
  LD %I5.1
  ST %MW10:X1
  // as ST:
  //   %MW10:X1 := %I5.1;

// Rung 154
  LD %I7.2
  ST %MW10:X2
  // as ST:
  //   %MW10:X2 := %I7.2;
  (* the ladder stored for this rung does not match its IL; not drawn *)

// Rung 155
  LD %I7.3
  ST %MW10:X3
  // as ST:
  //   %MW10:X3 := %I7.3;
  (* the ladder stored for this rung does not match its IL; not drawn *)

// Rung 156
  LD %I7.4
  ST %MW10:X4
  // as ST:
  //   %MW10:X4 := %I7.4;
  (* the ladder stored for this rung does not match its IL; not drawn *)

// Rung 157
  LD %I7.5
  ST %MW10:X5
  // as ST:
  //   %MW10:X5 := %I7.5;
  (* the ladder stored for this rung does not match its IL; not drawn *)

// Rung 158
  LD %I7.6
  ST %MW10:X6
  // as ST:
  //   %MW10:X6 := %I7.6;
  (* the ladder stored for this rung does not match its IL; not drawn *)

// Rung 159
  LD %I7.7
  ST %MW10:X7
  // as ST:
  //   %MW10:X7 := %I7.7;
  (* the ladder stored for this rung does not match its IL; not drawn *)

// Rung 160
  LD %M3
  ST %MW10:X8
  // as ST:
  //   %MW10:X8 := %M3;

// Rung 161
  LD %I7.9
  ST %MW10:X9
  // as ST:
  //   %MW10:X9 := %I7.9;
  (* the ladder stored for this rung does not match its IL; not drawn *)

// Rung 162
  LD %I7.10
  ST %MW10:X10
  // as ST:
  //   %MW10:X10 := %I7.10;
  (* the ladder stored for this rung does not match its IL; not drawn *)

// Rung 163
  LD %I7.11
  ST %MW10:X11
  // as ST:
  //   %MW10:X11 := %I7.11;
  (* the ladder stored for this rung does not match its IL; not drawn *)

// Rung 164
  LD %I7.12
  ST %MW10:X12
  // as ST:
  //   %MW10:X12 := %I7.12;
  (* the ladder stored for this rung does not match its IL; not drawn *)

// Rung 165
  LD %I7.13
  ST %MW10:X13
  // as ST:
  //   %MW10:X13 := %I7.13;
  (* the ladder stored for this rung does not match its IL; not drawn *)

// Rung 166
  LD %I7.14
  ST %MW10:X14
  // as ST:
  //   %MW10:X14 := %I7.14;
  (* the ladder stored for this rung does not match its IL; not drawn *)

// Rung 167
  LD %I7.15
  ST %MW10:X15
  // as ST:
  //   %MW10:X15 := %I7.15;
  (* the ladder stored for this rung does not match its IL; not drawn *)

// Rung 168
  LD %I7.16
  ST %MW11:X0
  // as ST:
  //   %MW11:X0 := %I7.16;
  (* the ladder stored for this rung does not match its IL; not drawn *)

// Rung 169
  LD %I7.17
  ST %MW11:X1
  // as ST:
  //   %MW11:X1 := %I7.17;
  (* the ladder stored for this rung does not match its IL; not drawn *)

// Rung 170
  LD %I7.18
  ST %MW11:X2
  // as ST:
  //   %MW11:X2 := %I7.18;
  (* the ladder stored for this rung does not match its IL; not drawn *)

// Rung 171
  LD %I7.19
  ST %MW11:X3
  // as ST:
  //   %MW11:X3 := %I7.19;
  (* the ladder stored for this rung does not match its IL; not drawn *)

// Rung 172
  LD %I7.20
  ST %MW11:X4
  // as ST:
  //   %MW11:X4 := %I7.20;
  (* the ladder stored for this rung does not match its IL; not drawn *)

// Rung 173
  LD %I7.21
  ST %MW11:X5
  // as ST:
  //   %MW11:X5 := %I7.21;
  (* the ladder stored for this rung does not match its IL; not drawn *)

// Rung 174
  LD %I7.22
  ST %MW11:X6
  // as ST:
  //   %MW11:X6 := %I7.22;
  (* the ladder stored for this rung does not match its IL; not drawn *)

// Rung 175
  LD %I7.23
  ST %MW11:X7
  // as ST:
  //   %MW11:X7 := %I7.23;
  (* the ladder stored for this rung does not match its IL; not drawn *)

// Rung 176
  LD %I7.24
  ST %MW11:X8
  // as ST:
  //   %MW11:X8 := %I7.24;
  (* the ladder stored for this rung does not match its IL; not drawn *)

// Rung 177
  LD %I7.25
  ST %MW11:X9
  // as ST:
  //   %MW11:X9 := %I7.25;
  (* the ladder stored for this rung does not match its IL; not drawn *)

// Rung 178
  LD %I7.26
  ST %MW11:X10
  // as ST:
  //   %MW11:X10 := %I7.26;
  (* the ladder stored for this rung does not match its IL; not drawn *)

// Rung 179
  LD %I7.27
  ST %MW11:X11
  // as ST:
  //   %MW11:X11 := %I7.27;
  (* the ladder stored for this rung does not match its IL; not drawn *)

// Rung 180
  LD %I7.28
  ST %MW11:X12
  // as ST:
  //   %MW11:X12 := %I7.28;
  (* the ladder stored for this rung does not match its IL; not drawn *)

// Rung 181
  LD %I7.29
  ST %MW11:X13
  // as ST:
  //   %MW11:X13 := %I7.29;
  (* the ladder stored for this rung does not match its IL; not drawn *)

// Rung 182
  LD %I7.30
  ST %MW11:X14
  // as ST:
  //   %MW11:X14 := %I7.30;
  (* the ladder stored for this rung does not match its IL; not drawn *)

// Rung 183
  LD %I7.31
  ST %MW11:X15
  // as ST:
  //   %MW11:X15 := %I7.31;
  (* the ladder stored for this rung does not match its IL; not drawn *)

POU Выходы 2.0
  (* SectionNumber=7 *)

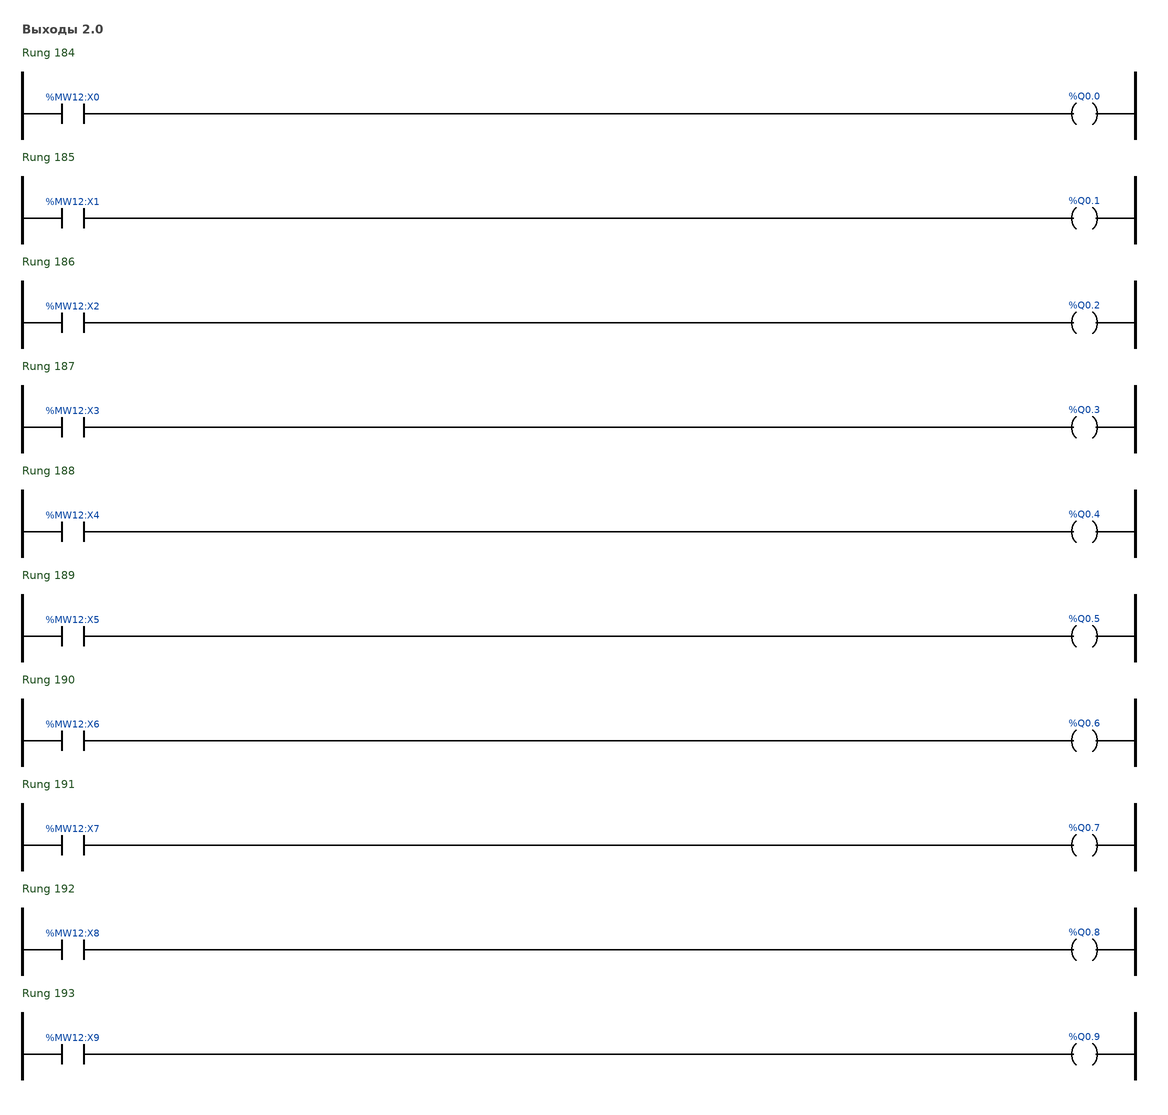

// Rung 184
  LD %MW12:X0
  ST %Q0.0
  // as ST:
  //   %Q0.0 := %MW12:X0;

// Rung 185
  LD %MW12:X1
  ST %Q0.1
  // as ST:
  //   %Q0.1 := %MW12:X1;

// Rung 186
  LD %MW12:X2
  ST %Q0.2
  // as ST:
  //   %Q0.2 := %MW12:X2;

// Rung 187
  LD %MW12:X3
  ST %Q0.3
  // as ST:
  //   %Q0.3 := %MW12:X3;

// Rung 188
  LD %MW12:X4
  ST %Q0.4
  // as ST:
  //   %Q0.4 := %MW12:X4;

// Rung 189
  LD %MW12:X5
  ST %Q0.5
  // as ST:
  //   %Q0.5 := %MW12:X5;

// Rung 190
  LD %MW12:X6
  ST %Q0.6
  // as ST:
  //   %Q0.6 := %MW12:X6;

// Rung 191
  LD %MW12:X7
  ST %Q0.7
  // as ST:
  //   %Q0.7 := %MW12:X7;

// Rung 192
  LD %MW12:X8
  ST %Q0.8
  // as ST:
  //   %Q0.8 := %MW12:X8;

// Rung 193
  LD %MW12:X9
  ST %Q0.9
  // as ST:
  //   %Q0.9 := %MW12:X9;

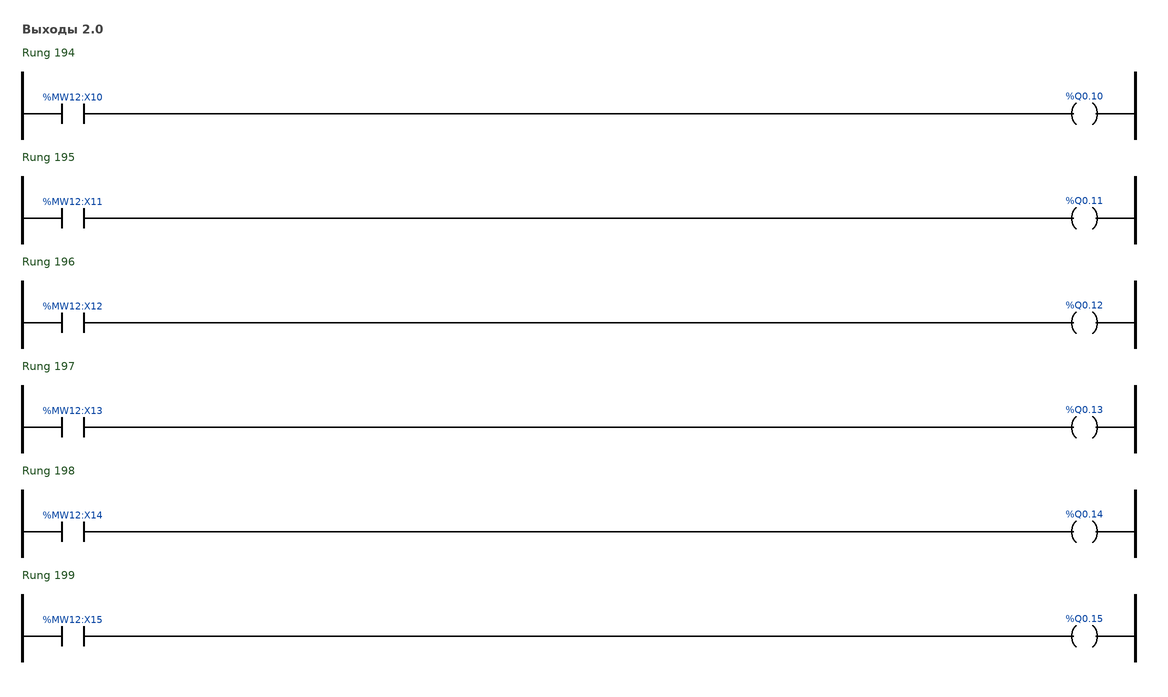

// Rung 194
  LD %MW12:X10
  ST %Q0.10
  // as ST:
  //   %Q0.10 := %MW12:X10;

// Rung 195
  LD %MW12:X11
  ST %Q0.11
  // as ST:
  //   %Q0.11 := %MW12:X11;

// Rung 196
  LD %MW12:X12
  ST %Q0.12
  // as ST:
  //   %Q0.12 := %MW12:X12;

// Rung 197
  LD %MW12:X13
  ST %Q0.13
  // as ST:
  //   %Q0.13 := %MW12:X13;

// Rung 198
  LD %MW12:X14
  ST %Q0.14
  // as ST:
  //   %Q0.14 := %MW12:X14;

// Rung 199
  LD %MW12:X15
  ST %Q0.15
  // as ST:
  //   %Q0.15 := %MW12:X15;

POU Выходы 2.6
  (* SectionNumber=8 *)

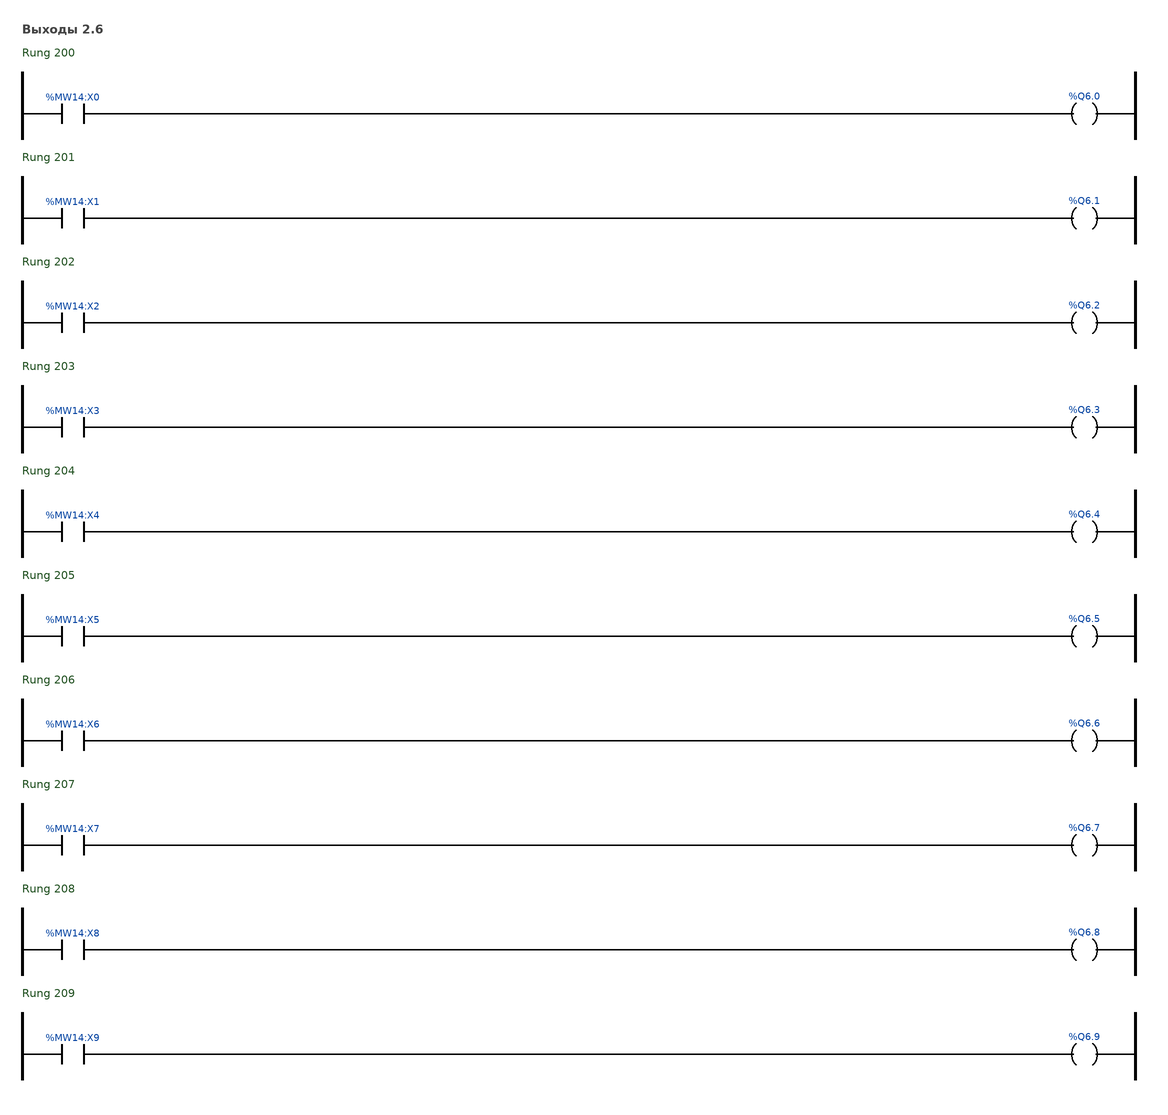

// Rung 200
  LD %MW14:X0
  ST %Q6.0
  // as ST:
  //   %Q6.0 := %MW14:X0;

// Rung 201
  LD %MW14:X1
  ST %Q6.1
  // as ST:
  //   %Q6.1 := %MW14:X1;

// Rung 202
  LD %MW14:X2
  ST %Q6.2
  // as ST:
  //   %Q6.2 := %MW14:X2;

// Rung 203
  LD %MW14:X3
  ST %Q6.3
  // as ST:
  //   %Q6.3 := %MW14:X3;

// Rung 204
  LD %MW14:X4
  ST %Q6.4
  // as ST:
  //   %Q6.4 := %MW14:X4;

// Rung 205
  LD %MW14:X5
  ST %Q6.5
  // as ST:
  //   %Q6.5 := %MW14:X5;

// Rung 206
  LD %MW14:X6
  ST %Q6.6
  // as ST:
  //   %Q6.6 := %MW14:X6;

// Rung 207
  LD %MW14:X7
  ST %Q6.7
  // as ST:
  //   %Q6.7 := %MW14:X7;

// Rung 208
  LD %MW14:X8
  ST %Q6.8
  // as ST:
  //   %Q6.8 := %MW14:X8;

// Rung 209
  LD %MW14:X9
  ST %Q6.9
  // as ST:
  //   %Q6.9 := %MW14:X9;

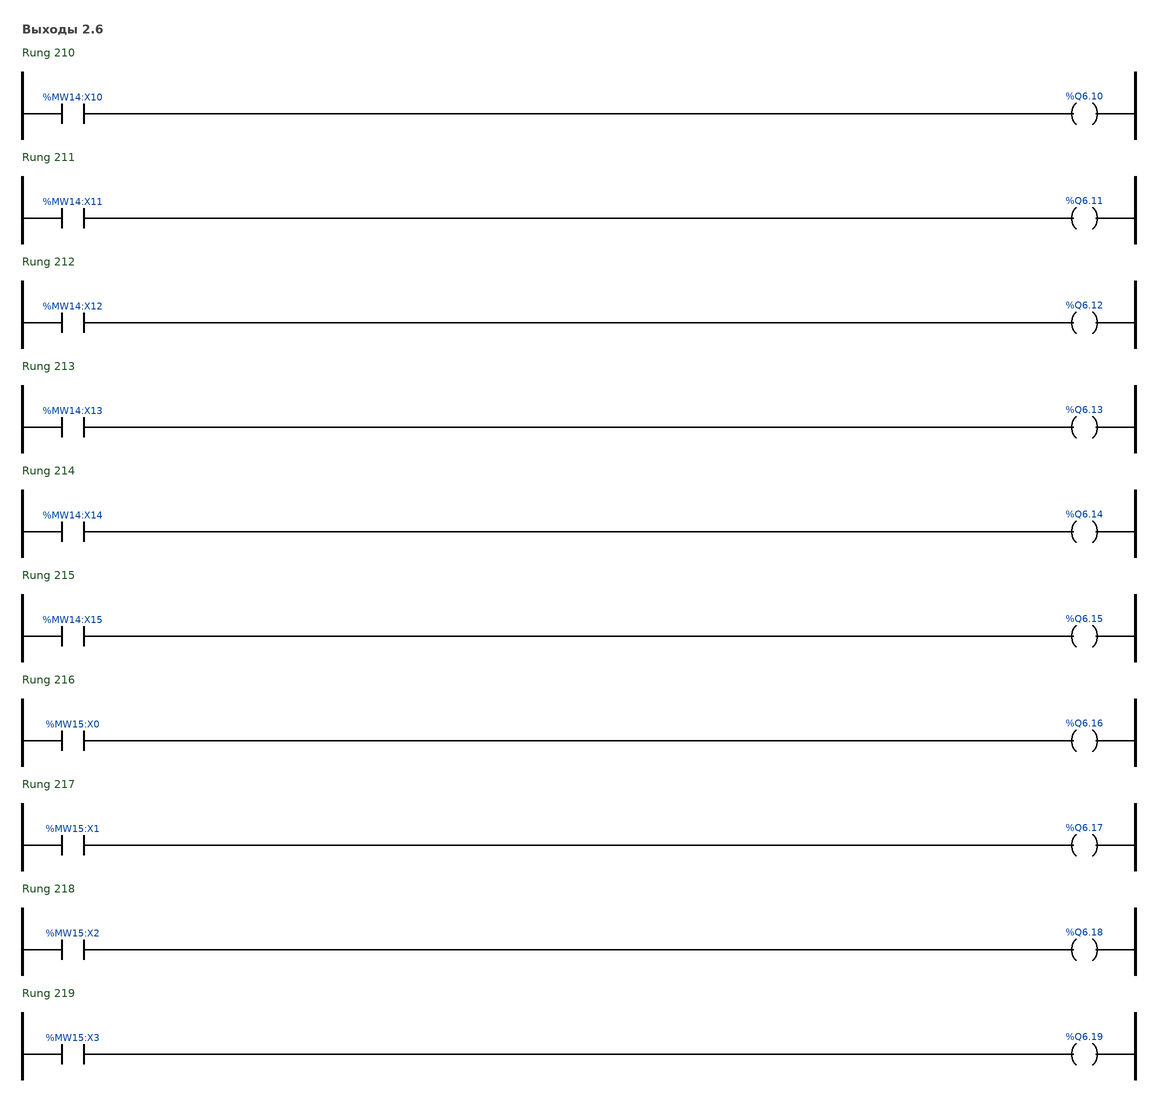

// Rung 210
  LD %MW14:X10
  ST %Q6.10
  // as ST:
  //   %Q6.10 := %MW14:X10;

// Rung 211
  LD %MW14:X11
  ST %Q6.11
  // as ST:
  //   %Q6.11 := %MW14:X11;

// Rung 212
  LD %MW14:X12
  ST %Q6.12
  // as ST:
  //   %Q6.12 := %MW14:X12;

// Rung 213
  LD %MW14:X13
  ST %Q6.13
  // as ST:
  //   %Q6.13 := %MW14:X13;

// Rung 214
  LD %MW14:X14
  ST %Q6.14
  // as ST:
  //   %Q6.14 := %MW14:X14;

// Rung 215
  LD %MW14:X15
  ST %Q6.15
  // as ST:
  //   %Q6.15 := %MW14:X15;

// Rung 216
  LD %MW15:X0
  ST %Q6.16
  // as ST:
  //   %Q6.16 := %MW15:X0;

// Rung 217
  LD %MW15:X1
  ST %Q6.17
  // as ST:
  //   %Q6.17 := %MW15:X1;

// Rung 218
  LD %MW15:X2
  ST %Q6.18
  // as ST:
  //   %Q6.18 := %MW15:X2;

// Rung 219
  LD %MW15:X3
  ST %Q6.19
  // as ST:
  //   %Q6.19 := %MW15:X3;

